    "phi" := "phi" + "w0c_11_24_5" * SIN(5 * 0.4 * "x") + "w0d_11_24_5" * COS(5 * 0.4 * "x");
    "phi" := "phi" + "w0c_11_24_6" * SIN(6 * 0.4 * "x") + "w0d_11_24_6" * COS(6 * 0.4 * "x");
    "acc" := "acc" + "phi";
    "x" := "feat_25";
    "phi" := "w0b_11_25" * "x" / (1.0 + EXP(-"x"));
    "phi" := "phi" + "w0c_11_25_1" * SIN(1 * 0.4 * "x") + "w0d_11_25_1" * COS(1 * 0.4 * "x");
    "phi" := "phi" + "w0c_11_25_2" * SIN(2 * 0.4 * "x") + "w0d_11_25_2" * COS(2 * 0.4 * "x");
    "phi" := "phi" + "w0c_11_25_3" * SIN(3 * 0.4 * "x") + "w0d_11_25_3" * COS(3 * 0.4 * "x");
    "phi" := "phi" + "w0c_11_25_4" * SIN(4 * 0.4 * "x") + "w0d_11_25_4" * COS(4 * 0.4 * "x");
    "phi" := "phi" + "w0c_11_25_5" * SIN(5 * 0.4 * "x") + "w0d_11_25_5" * COS(5 * 0.4 * "x");
    "phi" := "phi" + "w0c_11_25_6" * SIN(6 * 0.4 * "x") + "w0d_11_25_6" * COS(6 * 0.4 * "x");
    "acc" := "acc" + "phi";
    "x" := "feat_26";
    "phi" := "w0b_11_26" * "x" / (1.0 + EXP(-"x"));
    "phi" := "phi" + "w0c_11_26_1" * SIN(1 * 0.4 * "x") + "w0d_11_26_1" * COS(1 * 0.4 * "x");
    "phi" := "phi" + "w0c_11_26_2" * SIN(2 * 0.4 * "x") + "w0d_11_26_2" * COS(2 * 0.4 * "x");
    "phi" := "phi" + "w0c_11_26_3" * SIN(3 * 0.4 * "x") + "w0d_11_26_3" * COS(3 * 0.4 * "x");
    "phi" := "phi" + "w0c_11_26_4" * SIN(4 * 0.4 * "x") + "w0d_11_26_4" * COS(4 * 0.4 * "x");
    "phi" := "phi" + "w0c_11_26_5" * SIN(5 * 0.4 * "x") + "w0d_11_26_5" * COS(5 * 0.4 * "x");
    "phi" := "phi" + "w0c_11_26_6" * SIN(6 * 0.4 * "x") + "w0d_11_26_6" * COS(6 * 0.4 * "x");
    "acc" := "acc" + "phi";
    "x" := "feat_27";
    "phi" := "w0b_11_27" * "x" / (1.0 + EXP(-"x"));
    "phi" := "phi" + "w0c_11_27_1" * SIN(1 * 0.4 * "x") + "w0d_11_27_1" * COS(1 * 0.4 * "x");
    "phi" := "phi" + "w0c_11_27_2" * SIN(2 * 0.4 * "x") + "w0d_11_27_2" * COS(2 * 0.4 * "x");
    "phi" := "phi" + "w0c_11_27_3" * SIN(3 * 0.4 * "x") + "w0d_11_27_3" * COS(3 * 0.4 * "x");
    "phi" := "phi" + "w0c_11_27_4" * SIN(4 * 0.4 * "x") + "w0d_11_27_4" * COS(4 * 0.4 * "x");
    "phi" := "phi" + "w0c_11_27_5" * SIN(5 * 0.4 * "x") + "w0d_11_27_5" * COS(5 * 0.4 * "x");
    "phi" := "phi" + "w0c_11_27_6" * SIN(6 * 0.4 * "x") + "w0d_11_27_6" * COS(6 * 0.4 * "x");
    "acc" := "acc" + "phi";
    "x" := "feat_28";
    "phi" := "w0b_11_28" * "x" / (1.0 + EXP(-"x"));
    "phi" := "phi" + "w0c_11_28_1" * SIN(1 * 0.4 * "x") + "w0d_11_28_1" * COS(1 * 0.4 * "x");
    "phi" := "phi" + "w0c_11_28_2" * SIN(2 * 0.4 * "x") + "w0d_11_28_2" * COS(2 * 0.4 * "x");
    "phi" := "phi" + "w0c_11_28_3" * SIN(3 * 0.4 * "x") + "w0d_11_28_3" * COS(3 * 0.4 * "x");
    "phi" := "phi" + "w0c_11_28_4" * SIN(4 * 0.4 * "x") + "w0d_11_28_4" * COS(4 * 0.4 * "x");
    "phi" := "phi" + "w0c_11_28_5" * SIN(5 * 0.4 * "x") + "w0d_11_28_5" * COS(5 * 0.4 * "x");
    "phi" := "phi" + "w0c_11_28_6" * SIN(6 * 0.4 * "x") + "w0d_11_28_6" * COS(6 * 0.4 * "x");
    "acc" := "acc" + "phi";
    "h1_11" := "acc" + "b0_11";
    "acc" := 0.0;
    "x" := "feat_1";
    "phi" := "w0b_12_1" * "x" / (1.0 + EXP(-"x"));
    "phi" := "phi" + "w0c_12_1_1" * SIN(1 * 0.4 * "x") + "w0d_12_1_1" * COS(1 * 0.4 * "x");
    "phi" := "phi" + "w0c_12_1_2" * SIN(2 * 0.4 * "x") + "w0d_12_1_2" * COS(2 * 0.4 * "x");
    "phi" := "phi" + "w0c_12_1_3" * SIN(3 * 0.4 * "x") + "w0d_12_1_3" * COS(3 * 0.4 * "x");
    "phi" := "phi" + "w0c_12_1_4" * SIN(4 * 0.4 * "x") + "w0d_12_1_4" * COS(4 * 0.4 * "x");
    "phi" := "phi" + "w0c_12_1_5" * SIN(5 * 0.4 * "x") + "w0d_12_1_5" * COS(5 * 0.4 * "x");
    "phi" := "phi" + "w0c_12_1_6" * SIN(6 * 0.4 * "x") + "w0d_12_1_6" * COS(6 * 0.4 * "x");
    "acc" := "acc" + "phi";
    "x" := "feat_2";
    "phi" := "w0b_12_2" * "x" / (1.0 + EXP(-"x"));
    "phi" := "phi" + "w0c_12_2_1" * SIN(1 * 0.4 * "x") + "w0d_12_2_1" * COS(1 * 0.4 * "x");
    "phi" := "phi" + "w0c_12_2_2" * SIN(2 * 0.4 * "x") + "w0d_12_2_2" * COS(2 * 0.4 * "x");
    "phi" := "phi" + "w0c_12_2_3" * SIN(3 * 0.4 * "x") + "w0d_12_2_3" * COS(3 * 0.4 * "x");
    "phi" := "phi" + "w0c_12_2_4" * SIN(4 * 0.4 * "x") + "w0d_12_2_4" * COS(4 * 0.4 * "x");
    "phi" := "phi" + "w0c_12_2_5" * SIN(5 * 0.4 * "x") + "w0d_12_2_5" * COS(5 * 0.4 * "x");
    "phi" := "phi" + "w0c_12_2_6" * SIN(6 * 0.4 * "x") + "w0d_12_2_6" * COS(6 * 0.4 * "x");
    "acc" := "acc" + "phi";
    "x" := "feat_3";
    "phi" := "w0b_12_3" * "x" / (1.0 + EXP(-"x"));
    "phi" := "phi" + "w0c_12_3_1" * SIN(1 * 0.4 * "x") + "w0d_12_3_1" * COS(1 * 0.4 * "x");
    "phi" := "phi" + "w0c_12_3_2" * SIN(2 * 0.4 * "x") + "w0d_12_3_2" * COS(2 * 0.4 * "x");
    "phi" := "phi" + "w0c_12_3_3" * SIN(3 * 0.4 * "x") + "w0d_12_3_3" * COS(3 * 0.4 * "x");
    "phi" := "phi" + "w0c_12_3_4" * SIN(4 * 0.4 * "x") + "w0d_12_3_4" * COS(4 * 0.4 * "x");
    "phi" := "phi" + "w0c_12_3_5" * SIN(5 * 0.4 * "x") + "w0d_12_3_5" * COS(5 * 0.4 * "x");
    "phi" := "phi" + "w0c_12_3_6" * SIN(6 * 0.4 * "x") + "w0d_12_3_6" * COS(6 * 0.4 * "x");
    "acc" := "acc" + "phi";
    "x" := "feat_4";
    "phi" := "w0b_12_4" * "x" / (1.0 + EXP(-"x"));
    "phi" := "phi" + "w0c_12_4_1" * SIN(1 * 0.4 * "x") + "w0d_12_4_1" * COS(1 * 0.4 * "x");
    "phi" := "phi" + "w0c_12_4_2" * SIN(2 * 0.4 * "x") + "w0d_12_4_2" * COS(2 * 0.4 * "x");
    "phi" := "phi" + "w0c_12_4_3" * SIN(3 * 0.4 * "x") + "w0d_12_4_3" * COS(3 * 0.4 * "x");
    "phi" := "phi" + "w0c_12_4_4" * SIN(4 * 0.4 * "x") + "w0d_12_4_4" * COS(4 * 0.4 * "x");
    "phi" := "phi" + "w0c_12_4_5" * SIN(5 * 0.4 * "x") + "w0d_12_4_5" * COS(5 * 0.4 * "x");
    "phi" := "phi" + "w0c_12_4_6" * SIN(6 * 0.4 * "x") + "w0d_12_4_6" * COS(6 * 0.4 * "x");
    "acc" := "acc" + "phi";
    "x" := "feat_5";
    "phi" := "w0b_12_5" * "x" / (1.0 + EXP(-"x"));
    "phi" := "phi" + "w0c_12_5_1" * SIN(1 * 0.4 * "x") + "w0d_12_5_1" * COS(1 * 0.4 * "x");
    "phi" := "phi" + "w0c_12_5_2" * SIN(2 * 0.4 * "x") + "w0d_12_5_2" * COS(2 * 0.4 * "x");
    "phi" := "phi" + "w0c_12_5_3" * SIN(3 * 0.4 * "x") + "w0d_12_5_3" * COS(3 * 0.4 * "x");
    "phi" := "phi" + "w0c_12_5_4" * SIN(4 * 0.4 * "x") + "w0d_12_5_4" * COS(4 * 0.4 * "x");
    "phi" := "phi" + "w0c_12_5_5" * SIN(5 * 0.4 * "x") + "w0d_12_5_5" * COS(5 * 0.4 * "x");
    "phi" := "phi" + "w0c_12_5_6" * SIN(6 * 0.4 * "x") + "w0d_12_5_6" * COS(6 * 0.4 * "x");
    "acc" := "acc" + "phi";
    "x" := "feat_6";
    "phi" := "w0b_12_6" * "x" / (1.0 + EXP(-"x"));
    "phi" := "phi" + "w0c_12_6_1" * SIN(1 * 0.4 * "x") + "w0d_12_6_1" * COS(1 * 0.4 * "x");
    "phi" := "phi" + "w0c_12_6_2" * SIN(2 * 0.4 * "x") + "w0d_12_6_2" * COS(2 * 0.4 * "x");
    "phi" := "phi" + "w0c_12_6_3" * SIN(3 * 0.4 * "x") + "w0d_12_6_3" * COS(3 * 0.4 * "x");
    "phi" := "phi" + "w0c_12_6_4" * SIN(4 * 0.4 * "x") + "w0d_12_6_4" * COS(4 * 0.4 * "x");
    "phi" := "phi" + "w0c_12_6_5" * SIN(5 * 0.4 * "x") + "w0d_12_6_5" * COS(5 * 0.4 * "x");
    "phi" := "phi" + "w0c_12_6_6" * SIN(6 * 0.4 * "x") + "w0d_12_6_6" * COS(6 * 0.4 * "x");
    "acc" := "acc" + "phi";
    "x" := "feat_7";
    "phi" := "w0b_12_7" * "x" / (1.0 + EXP(-"x"));
    "phi" := "phi" + "w0c_12_7_1" * SIN(1 * 0.4 * "x") + "w0d_12_7_1" * COS(1 * 0.4 * "x");
    "phi" := "phi" + "w0c_12_7_2" * SIN(2 * 0.4 * "x") + "w0d_12_7_2" * COS(2 * 0.4 * "x");
    "phi" := "phi" + "w0c_12_7_3" * SIN(3 * 0.4 * "x") + "w0d_12_7_3" * COS(3 * 0.4 * "x");
    "phi" := "phi" + "w0c_12_7_4" * SIN(4 * 0.4 * "x") + "w0d_12_7_4" * COS(4 * 0.4 * "x");
    "phi" := "phi" + "w0c_12_7_5" * SIN(5 * 0.4 * "x") + "w0d_12_7_5" * COS(5 * 0.4 * "x");
    "phi" := "phi" + "w0c_12_7_6" * SIN(6 * 0.4 * "x") + "w0d_12_7_6" * COS(6 * 0.4 * "x");
    "acc" := "acc" + "phi";
    "x" := "feat_8";
    "phi" := "w0b_12_8" * "x" / (1.0 + EXP(-"x"));
    "phi" := "phi" + "w0c_12_8_1" * SIN(1 * 0.4 * "x") + "w0d_12_8_1" * COS(1 * 0.4 * "x");
    "phi" := "phi" + "w0c_12_8_2" * SIN(2 * 0.4 * "x") + "w0d_12_8_2" * COS(2 * 0.4 * "x");
    "phi" := "phi" + "w0c_12_8_3" * SIN(3 * 0.4 * "x") + "w0d_12_8_3" * COS(3 * 0.4 * "x");
    "phi" := "phi" + "w0c_12_8_4" * SIN(4 * 0.4 * "x") + "w0d_12_8_4" * COS(4 * 0.4 * "x");
    "phi" := "phi" + "w0c_12_8_5" * SIN(5 * 0.4 * "x") + "w0d_12_8_5" * COS(5 * 0.4 * "x");
    "phi" := "phi" + "w0c_12_8_6" * SIN(6 * 0.4 * "x") + "w0d_12_8_6" * COS(6 * 0.4 * "x");
    "acc" := "acc" + "phi";
    "x" := "feat_9";
    "phi" := "w0b_12_9" * "x" / (1.0 + EXP(-"x"));
    "phi" := "phi" + "w0c_12_9_1" * SIN(1 * 0.4 * "x") + "w0d_12_9_1" * COS(1 * 0.4 * "x");
    "phi" := "phi" + "w0c_12_9_2" * SIN(2 * 0.4 * "x") + "w0d_12_9_2" * COS(2 * 0.4 * "x");
    "phi" := "phi" + "w0c_12_9_3" * SIN(3 * 0.4 * "x") + "w0d_12_9_3" * COS(3 * 0.4 * "x");
    "phi" := "phi" + "w0c_12_9_4" * SIN(4 * 0.4 * "x") + "w0d_12_9_4" * COS(4 * 0.4 * "x");
    "phi" := "phi" + "w0c_12_9_5" * SIN(5 * 0.4 * "x") + "w0d_12_9_5" * COS(5 * 0.4 * "x");
    "phi" := "phi" + "w0c_12_9_6" * SIN(6 * 0.4 * "x") + "w0d_12_9_6" * COS(6 * 0.4 * "x");
    "acc" := "acc" + "phi";
    "x" := "feat_10";
    "phi" := "w0b_12_10" * "x" / (1.0 + EXP(-"x"));
    "phi" := "phi" + "w0c_12_10_1" * SIN(1 * 0.4 * "x") + "w0d_12_10_1" * COS(1 * 0.4 * "x");
    "phi" := "phi" + "w0c_12_10_2" * SIN(2 * 0.4 * "x") + "w0d_12_10_2" * COS(2 * 0.4 * "x");
    "phi" := "phi" + "w0c_12_10_3" * SIN(3 * 0.4 * "x") + "w0d_12_10_3" * COS(3 * 0.4 * "x");
    "phi" := "phi" + "w0c_12_10_4" * SIN(4 * 0.4 * "x") + "w0d_12_10_4" * COS(4 * 0.4 * "x");
    "phi" := "phi" + "w0c_12_10_5" * SIN(5 * 0.4 * "x") + "w0d_12_10_5" * COS(5 * 0.4 * "x");
    "phi" := "phi" + "w0c_12_10_6" * SIN(6 * 0.4 * "x") + "w0d_12_10_6" * COS(6 * 0.4 * "x");
    "acc" := "acc" + "phi";
    "x" := "feat_11";
    "phi" := "w0b_12_11" * "x" / (1.0 + EXP(-"x"));
    "phi" := "phi" + "w0c_12_11_1" * SIN(1 * 0.4 * "x") + "w0d_12_11_1" * COS(1 * 0.4 * "x");
    "phi" := "phi" + "w0c_12_11_2" * SIN(2 * 0.4 * "x") + "w0d_12_11_2" * COS(2 * 0.4 * "x");
    "phi" := "phi" + "w0c_12_11_3" * SIN(3 * 0.4 * "x") + "w0d_12_11_3" * COS(3 * 0.4 * "x");
    "phi" := "phi" + "w0c_12_11_4" * SIN(4 * 0.4 * "x") + "w0d_12_11_4" * COS(4 * 0.4 * "x");
    "phi" := "phi" + "w0c_12_11_5" * SIN(5 * 0.4 * "x") + "w0d_12_11_5" * COS(5 * 0.4 * "x");
    "phi" := "phi" + "w0c_12_11_6" * SIN(6 * 0.4 * "x") + "w0d_12_11_6" * COS(6 * 0.4 * "x");
    "acc" := "acc" + "phi";
    "x" := "feat_12";
    "phi" := "w0b_12_12" * "x" / (1.0 + EXP(-"x"));
    "phi" := "phi" + "w0c_12_12_1" * SIN(1 * 0.4 * "x") + "w0d_12_12_1" * COS(1 * 0.4 * "x");
    "phi" := "phi" + "w0c_12_12_2" * SIN(2 * 0.4 * "x") + "w0d_12_12_2" * COS(2 * 0.4 * "x");
    "phi" := "phi" + "w0c_12_12_3" * SIN(3 * 0.4 * "x") + "w0d_12_12_3" * COS(3 * 0.4 * "x");
    "phi" := "phi" + "w0c_12_12_4" * SIN(4 * 0.4 * "x") + "w0d_12_12_4" * COS(4 * 0.4 * "x");
    "phi" := "phi" + "w0c_12_12_5" * SIN(5 * 0.4 * "x") + "w0d_12_12_5" * COS(5 * 0.4 * "x");
    "phi" := "phi" + "w0c_12_12_6" * SIN(6 * 0.4 * "x") + "w0d_12_12_6" * COS(6 * 0.4 * "x");
    "acc" := "acc" + "phi";
    "x" := "feat_13";
    "phi" := "w0b_12_13" * "x" / (1.0 + EXP(-"x"));
    "phi" := "phi" + "w0c_12_13_1" * SIN(1 * 0.4 * "x") + "w0d_12_13_1" * COS(1 * 0.4 * "x");
    "phi" := "phi" + "w0c_12_13_2" * SIN(2 * 0.4 * "x") + "w0d_12_13_2" * COS(2 * 0.4 * "x");
    "phi" := "phi" + "w0c_12_13_3" * SIN(3 * 0.4 * "x") + "w0d_12_13_3" * COS(3 * 0.4 * "x");
    "phi" := "phi" + "w0c_12_13_4" * SIN(4 * 0.4 * "x") + "w0d_12_13_4" * COS(4 * 0.4 * "x");
    "phi" := "phi" + "w0c_12_13_5" * SIN(5 * 0.4 * "x") + "w0d_12_13_5" * COS(5 * 0.4 * "x");
    "phi" := "phi" + "w0c_12_13_6" * SIN(6 * 0.4 * "x") + "w0d_12_13_6" * COS(6 * 0.4 * "x");
    "acc" := "acc" + "phi";
    "x" := "feat_14";
    "phi" := "w0b_12_14" * "x" / (1.0 + EXP(-"x"));
    "phi" := "phi" + "w0c_12_14_1" * SIN(1 * 0.4 * "x") + "w0d_12_14_1" * COS(1 * 0.4 * "x");
    "phi" := "phi" + "w0c_12_14_2" * SIN(2 * 0.4 * "x") + "w0d_12_14_2" * COS(2 * 0.4 * "x");
    "phi" := "phi" + "w0c_12_14_3" * SIN(3 * 0.4 * "x") + "w0d_12_14_3" * COS(3 * 0.4 * "x");
    "phi" := "phi" + "w0c_12_14_4" * SIN(4 * 0.4 * "x") + "w0d_12_14_4" * COS(4 * 0.4 * "x");
    "phi" := "phi" + "w0c_12_14_5" * SIN(5 * 0.4 * "x") + "w0d_12_14_5" * COS(5 * 0.4 * "x");
    "phi" := "phi" + "w0c_12_14_6" * SIN(6 * 0.4 * "x") + "w0d_12_14_6" * COS(6 * 0.4 * "x");
    "acc" := "acc" + "phi";
    "x" := "feat_15";
    "phi" := "w0b_12_15" * "x" / (1.0 + EXP(-"x"));
    "phi" := "phi" + "w0c_12_15_1" * SIN(1 * 0.4 * "x") + "w0d_12_15_1" * COS(1 * 0.4 * "x");
    "phi" := "phi" + "w0c_12_15_2" * SIN(2 * 0.4 * "x") + "w0d_12_15_2" * COS(2 * 0.4 * "x");
    "phi" := "phi" + "w0c_12_15_3" * SIN(3 * 0.4 * "x") + "w0d_12_15_3" * COS(3 * 0.4 * "x");
    "phi" := "phi" + "w0c_12_15_4" * SIN(4 * 0.4 * "x") + "w0d_12_15_4" * COS(4 * 0.4 * "x");
    "phi" := "phi" + "w0c_12_15_5" * SIN(5 * 0.4 * "x") + "w0d_12_15_5" * COS(5 * 0.4 * "x");
    "phi" := "phi" + "w0c_12_15_6" * SIN(6 * 0.4 * "x") + "w0d_12_15_6" * COS(6 * 0.4 * "x");
    "acc" := "acc" + "phi";
    "x" := "feat_16";
    "phi" := "w0b_12_16" * "x" / (1.0 + EXP(-"x"));
    "phi" := "phi" + "w0c_12_16_1" * SIN(1 * 0.4 * "x") + "w0d_12_16_1" * COS(1 * 0.4 * "x");
    "phi" := "phi" + "w0c_12_16_2" * SIN(2 * 0.4 * "x") + "w0d_12_16_2" * COS(2 * 0.4 * "x");
    "phi" := "phi" + "w0c_12_16_3" * SIN(3 * 0.4 * "x") + "w0d_12_16_3" * COS(3 * 0.4 * "x");
    "phi" := "phi" + "w0c_12_16_4" * SIN(4 * 0.4 * "x") + "w0d_12_16_4" * COS(4 * 0.4 * "x");
    "phi" := "phi" + "w0c_12_16_5" * SIN(5 * 0.4 * "x") + "w0d_12_16_5" * COS(5 * 0.4 * "x");
    "phi" := "phi" + "w0c_12_16_6" * SIN(6 * 0.4 * "x") + "w0d_12_16_6" * COS(6 * 0.4 * "x");
    "acc" := "acc" + "phi";
    "x" := "feat_17";
    "phi" := "w0b_12_17" * "x" / (1.0 + EXP(-"x"));
    "phi" := "phi" + "w0c_12_17_1" * SIN(1 * 0.4 * "x") + "w0d_12_17_1" * COS(1 * 0.4 * "x");
    "phi" := "phi" + "w0c_12_17_2" * SIN(2 * 0.4 * "x") + "w0d_12_17_2" * COS(2 * 0.4 * "x");
    "phi" := "phi" + "w0c_12_17_3" * SIN(3 * 0.4 * "x") + "w0d_12_17_3" * COS(3 * 0.4 * "x");
    "phi" := "phi" + "w0c_12_17_4" * SIN(4 * 0.4 * "x") + "w0d_12_17_4" * COS(4 * 0.4 * "x");
    "phi" := "phi" + "w0c_12_17_5" * SIN(5 * 0.4 * "x") + "w0d_12_17_5" * COS(5 * 0.4 * "x");
    "phi" := "phi" + "w0c_12_17_6" * SIN(6 * 0.4 * "x") + "w0d_12_17_6" * COS(6 * 0.4 * "x");
    "acc" := "acc" + "phi";
    "x" := "feat_18";
    "phi" := "w0b_12_18" * "x" / (1.0 + EXP(-"x"));
    "phi" := "phi" + "w0c_12_18_1" * SIN(1 * 0.4 * "x") + "w0d_12_18_1" * COS(1 * 0.4 * "x");
    "phi" := "phi" + "w0c_12_18_2" * SIN(2 * 0.4 * "x") + "w0d_12_18_2" * COS(2 * 0.4 * "x");
    "phi" := "phi" + "w0c_12_18_3" * SIN(3 * 0.4 * "x") + "w0d_12_18_3" * COS(3 * 0.4 * "x");
    "phi" := "phi" + "w0c_12_18_4" * SIN(4 * 0.4 * "x") + "w0d_12_18_4" * COS(4 * 0.4 * "x");
    "phi" := "phi" + "w0c_12_18_5" * SIN(5 * 0.4 * "x") + "w0d_12_18_5" * COS(5 * 0.4 * "x");
    "phi" := "phi" + "w0c_12_18_6" * SIN(6 * 0.4 * "x") + "w0d_12_18_6" * COS(6 * 0.4 * "x");
    "acc" := "acc" + "phi";
    "x" := "feat_19";
    "phi" := "w0b_12_19" * "x" / (1.0 + EXP(-"x"));
    "phi" := "phi" + "w0c_12_19_1" * SIN(1 * 0.4 * "x") + "w0d_12_19_1" * COS(1 * 0.4 * "x");
    "phi" := "phi" + "w0c_12_19_2" * SIN(2 * 0.4 * "x") + "w0d_12_19_2" * COS(2 * 0.4 * "x");
    "phi" := "phi" + "w0c_12_19_3" * SIN(3 * 0.4 * "x") + "w0d_12_19_3" * COS(3 * 0.4 * "x");
    "phi" := "phi" + "w0c_12_19_4" * SIN(4 * 0.4 * "x") + "w0d_12_19_4" * COS(4 * 0.4 * "x");
    "phi" := "phi" + "w0c_12_19_5" * SIN(5 * 0.4 * "x") + "w0d_12_19_5" * COS(5 * 0.4 * "x");
    "phi" := "phi" + "w0c_12_19_6" * SIN(6 * 0.4 * "x") + "w0d_12_19_6" * COS(6 * 0.4 * "x");
    "acc" := "acc" + "phi";
    "x" := "feat_20";
    "phi" := "w0b_12_20" * "x" / (1.0 + EXP(-"x"));
    "phi" := "phi" + "w0c_12_20_1" * SIN(1 * 0.4 * "x") + "w0d_12_20_1" * COS(1 * 0.4 * "x");
    "phi" := "phi" + "w0c_12_20_2" * SIN(2 * 0.4 * "x") + "w0d_12_20_2" * COS(2 * 0.4 * "x");
    "phi" := "phi" + "w0c_12_20_3" * SIN(3 * 0.4 * "x") + "w0d_12_20_3" * COS(3 * 0.4 * "x");
    "phi" := "phi" + "w0c_12_20_4" * SIN(4 * 0.4 * "x") + "w0d_12_20_4" * COS(4 * 0.4 * "x");
    "phi" := "phi" + "w0c_12_20_5" * SIN(5 * 0.4 * "x") + "w0d_12_20_5" * COS(5 * 0.4 * "x");
    "phi" := "phi" + "w0c_12_20_6" * SIN(6 * 0.4 * "x") + "w0d_12_20_6" * COS(6 * 0.4 * "x");
    "acc" := "acc" + "phi";
    "x" := "feat_21";
    "phi" := "w0b_12_21" * "x" / (1.0 + EXP(-"x"));
    "phi" := "phi" + "w0c_12_21_1" * SIN(1 * 0.4 * "x") + "w0d_12_21_1" * COS(1 * 0.4 * "x");
    "phi" := "phi" + "w0c_12_21_2" * SIN(2 * 0.4 * "x") + "w0d_12_21_2" * COS(2 * 0.4 * "x");
    "phi" := "phi" + "w0c_12_21_3" * SIN(3 * 0.4 * "x") + "w0d_12_21_3" * COS(3 * 0.4 * "x");
    "phi" := "phi" + "w0c_12_21_4" * SIN(4 * 0.4 * "x") + "w0d_12_21_4" * COS(4 * 0.4 * "x");
    "phi" := "phi" + "w0c_12_21_5" * SIN(5 * 0.4 * "x") + "w0d_12_21_5" * COS(5 * 0.4 * "x");
    "phi" := "phi" + "w0c_12_21_6" * SIN(6 * 0.4 * "x") + "w0d_12_21_6" * COS(6 * 0.4 * "x");
    "acc" := "acc" + "phi";
    "x" := "feat_22";
    "phi" := "w0b_12_22" * "x" / (1.0 + EXP(-"x"));
    "phi" := "phi" + "w0c_12_22_1" * SIN(1 * 0.4 * "x") + "w0d_12_22_1" * COS(1 * 0.4 * "x");
    "phi" := "phi" + "w0c_12_22_2" * SIN(2 * 0.4 * "x") + "w0d_12_22_2" * COS(2 * 0.4 * "x");
    "phi" := "phi" + "w0c_12_22_3" * SIN(3 * 0.4 * "x") + "w0d_12_22_3" * COS(3 * 0.4 * "x");
    "phi" := "phi" + "w0c_12_22_4" * SIN(4 * 0.4 * "x") + "w0d_12_22_4" * COS(4 * 0.4 * "x");
    "phi" := "phi" + "w0c_12_22_5" * SIN(5 * 0.4 * "x") + "w0d_12_22_5" * COS(5 * 0.4 * "x");
    "phi" := "phi" + "w0c_12_22_6" * SIN(6 * 0.4 * "x") + "w0d_12_22_6" * COS(6 * 0.4 * "x");
    "acc" := "acc" + "phi";
    "x" := "feat_23";
    "phi" := "w0b_12_23" * "x" / (1.0 + EXP(-"x"));
    "phi" := "phi" + "w0c_12_23_1" * SIN(1 * 0.4 * "x") + "w0d_12_23_1" * COS(1 * 0.4 * "x");
    "phi" := "phi" + "w0c_12_23_2" * SIN(2 * 0.4 * "x") + "w0d_12_23_2" * COS(2 * 0.4 * "x");
    "phi" := "phi" + "w0c_12_23_3" * SIN(3 * 0.4 * "x") + "w0d_12_23_3" * COS(3 * 0.4 * "x");
    "phi" := "phi" + "w0c_12_23_4" * SIN(4 * 0.4 * "x") + "w0d_12_23_4" * COS(4 * 0.4 * "x");
    "phi" := "phi" + "w0c_12_23_5" * SIN(5 * 0.4 * "x") + "w0d_12_23_5" * COS(5 * 0.4 * "x");
    "phi" := "phi" + "w0c_12_23_6" * SIN(6 * 0.4 * "x") + "w0d_12_23_6" * COS(6 * 0.4 * "x");
    "acc" := "acc" + "phi";
    "x" := "feat_24";
    "phi" := "w0b_12_24" * "x" / (1.0 + EXP(-"x"));
    "phi" := "phi" + "w0c_12_24_1" * SIN(1 * 0.4 * "x") + "w0d_12_24_1" * COS(1 * 0.4 * "x");
    "phi" := "phi" + "w0c_12_24_2" * SIN(2 * 0.4 * "x") + "w0d_12_24_2" * COS(2 * 0.4 * "x");
    "phi" := "phi" + "w0c_12_24_3" * SIN(3 * 0.4 * "x") + "w0d_12_24_3" * COS(3 * 0.4 * "x");
    "phi" := "phi" + "w0c_12_24_4" * SIN(4 * 0.4 * "x") + "w0d_12_24_4" * COS(4 * 0.4 * "x");
    "phi" := "phi" + "w0c_12_24_5" * SIN(5 * 0.4 * "x") + "w0d_12_24_5" * COS(5 * 0.4 * "x");
    "phi" := "phi" + "w0c_12_24_6" * SIN(6 * 0.4 * "x") + "w0d_12_24_6" * COS(6 * 0.4 * "x");
    "acc" := "acc" + "phi";
    "x" := "feat_25";
    "phi" := "w0b_12_25" * "x" / (1.0 + EXP(-"x"));
    "phi" := "phi" + "w0c_12_25_1" * SIN(1 * 0.4 * "x") + "w0d_12_25_1" * COS(1 * 0.4 * "x");
    "phi" := "phi" + "w0c_12_25_2" * SIN(2 * 0.4 * "x") + "w0d_12_25_2" * COS(2 * 0.4 * "x");
    "phi" := "phi" + "w0c_12_25_3" * SIN(3 * 0.4 * "x") + "w0d_12_25_3" * COS(3 * 0.4 * "x");
    "phi" := "phi" + "w0c_12_25_4" * SIN(4 * 0.4 * "x") + "w0d_12_25_4" * COS(4 * 0.4 * "x");
    "phi" := "phi" + "w0c_12_25_5" * SIN(5 * 0.4 * "x") + "w0d_12_25_5" * COS(5 * 0.4 * "x");
    "phi" := "phi" + "w0c_12_25_6" * SIN(6 * 0.4 * "x") + "w0d_12_25_6" * COS(6 * 0.4 * "x");
    "acc" := "acc" + "phi";
    "x" := "feat_26";
    "phi" := "w0b_12_26" * "x" / (1.0 + EXP(-"x"));
    "phi" := "phi" + "w0c_12_26_1" * SIN(1 * 0.4 * "x") + "w0d_12_26_1" * COS(1 * 0.4 * "x");
    "phi" := "phi" + "w0c_12_26_2" * SIN(2 * 0.4 * "x") + "w0d_12_26_2" * COS(2 * 0.4 * "x");
    "phi" := "phi" + "w0c_12_26_3" * SIN(3 * 0.4 * "x") + "w0d_12_26_3" * COS(3 * 0.4 * "x");
    "phi" := "phi" + "w0c_12_26_4" * SIN(4 * 0.4 * "x") + "w0d_12_26_4" * COS(4 * 0.4 * "x");
    "phi" := "phi" + "w0c_12_26_5" * SIN(5 * 0.4 * "x") + "w0d_12_26_5" * COS(5 * 0.4 * "x");
    "phi" := "phi" + "w0c_12_26_6" * SIN(6 * 0.4 * "x") + "w0d_12_26_6" * COS(6 * 0.4 * "x");
    "acc" := "acc" + "phi";
    "x" := "feat_27";
    "phi" := "w0b_12_27" * "x" / (1.0 + EXP(-"x"));
    "phi" := "phi" + "w0c_12_27_1" * SIN(1 * 0.4 * "x") + "w0d_12_27_1" * COS(1 * 0.4 * "x");
    "phi" := "phi" + "w0c_12_27_2" * SIN(2 * 0.4 * "x") + "w0d_12_27_2" * COS(2 * 0.4 * "x");
    "phi" := "phi" + "w0c_12_27_3" * SIN(3 * 0.4 * "x") + "w0d_12_27_3" * COS(3 * 0.4 * "x");
    "phi" := "phi" + "w0c_12_27_4" * SIN(4 * 0.4 * "x") + "w0d_12_27_4" * COS(4 * 0.4 * "x");
    "phi" := "phi" + "w0c_12_27_5" * SIN(5 * 0.4 * "x") + "w0d_12_27_5" * COS(5 * 0.4 * "x");
    "phi" := "phi" + "w0c_12_27_6" * SIN(6 * 0.4 * "x") + "w0d_12_27_6" * COS(6 * 0.4 * "x");
    "acc" := "acc" + "phi";
    "x" := "feat_28";
    "phi" := "w0b_12_28" * "x" / (1.0 + EXP(-"x"));
    "phi" := "phi" + "w0c_12_28_1" * SIN(1 * 0.4 * "x") + "w0d_12_28_1" * COS(1 * 0.4 * "x");
    "phi" := "phi" + "w0c_12_28_2" * SIN(2 * 0.4 * "x") + "w0d_12_28_2" * COS(2 * 0.4 * "x");
    "phi" := "phi" + "w0c_12_28_3" * SIN(3 * 0.4 * "x") + "w0d_12_28_3" * COS(3 * 0.4 * "x");
    "phi" := "phi" + "w0c_12_28_4" * SIN(4 * 0.4 * "x") + "w0d_12_28_4" * COS(4 * 0.4 * "x");
    "phi" := "phi" + "w0c_12_28_5" * SIN(5 * 0.4 * "x") + "w0d_12_28_5" * COS(5 * 0.4 * "x");
    "phi" := "phi" + "w0c_12_28_6" * SIN(6 * 0.4 * "x") + "w0d_12_28_6" * COS(6 * 0.4 * "x");
    "acc" := "acc" + "phi";
    "h1_12" := "acc" + "b0_12";
    "acc" := 0.0;
    "x" := "feat_1";
    "phi" := "w0b_13_1" * "x" / (1.0 + EXP(-"x"));
    "phi" := "phi" + "w0c_13_1_1" * SIN(1 * 0.4 * "x") + "w0d_13_1_1" * COS(1 * 0.4 * "x");
    "phi" := "phi" + "w0c_13_1_2" * SIN(2 * 0.4 * "x") + "w0d_13_1_2" * COS(2 * 0.4 * "x");
    "phi" := "phi" + "w0c_13_1_3" * SIN(3 * 0.4 * "x") + "w0d_13_1_3" * COS(3 * 0.4 * "x");
    "phi" := "phi" + "w0c_13_1_4" * SIN(4 * 0.4 * "x") + "w0d_13_1_4" * COS(4 * 0.4 * "x");
    "phi" := "phi" + "w0c_13_1_5" * SIN(5 * 0.4 * "x") + "w0d_13_1_5" * COS(5 * 0.4 * "x");
    "phi" := "phi" + "w0c_13_1_6" * SIN(6 * 0.4 * "x") + "w0d_13_1_6" * COS(6 * 0.4 * "x");
    "acc" := "acc" + "phi";
    "x" := "feat_2";
    "phi" := "w0b_13_2" * "x" / (1.0 + EXP(-"x"));
    "phi" := "phi" + "w0c_13_2_1" * SIN(1 * 0.4 * "x") + "w0d_13_2_1" * COS(1 * 0.4 * "x");
    "phi" := "phi" + "w0c_13_2_2" * SIN(2 * 0.4 * "x") + "w0d_13_2_2" * COS(2 * 0.4 * "x");
    "phi" := "phi" + "w0c_13_2_3" * SIN(3 * 0.4 * "x") + "w0d_13_2_3" * COS(3 * 0.4 * "x");
    "phi" := "phi" + "w0c_13_2_4" * SIN(4 * 0.4 * "x") + "w0d_13_2_4" * COS(4 * 0.4 * "x");
    "phi" := "phi" + "w0c_13_2_5" * SIN(5 * 0.4 * "x") + "w0d_13_2_5" * COS(5 * 0.4 * "x");
    "phi" := "phi" + "w0c_13_2_6" * SIN(6 * 0.4 * "x") + "w0d_13_2_6" * COS(6 * 0.4 * "x");
    "acc" := "acc" + "phi";
    "x" := "feat_3";
    "phi" := "w0b_13_3" * "x" / (1.0 + EXP(-"x"));
    "phi" := "phi" + "w0c_13_3_1" * SIN(1 * 0.4 * "x") + "w0d_13_3_1" * COS(1 * 0.4 * "x");
    "phi" := "phi" + "w0c_13_3_2" * SIN(2 * 0.4 * "x") + "w0d_13_3_2" * COS(2 * 0.4 * "x");
    "phi" := "phi" + "w0c_13_3_3" * SIN(3 * 0.4 * "x") + "w0d_13_3_3" * COS(3 * 0.4 * "x");
    "phi" := "phi" + "w0c_13_3_4" * SIN(4 * 0.4 * "x") + "w0d_13_3_4" * COS(4 * 0.4 * "x");
    "phi" := "phi" + "w0c_13_3_5" * SIN(5 * 0.4 * "x") + "w0d_13_3_5" * COS(5 * 0.4 * "x");
    "phi" := "phi" + "w0c_13_3_6" * SIN(6 * 0.4 * "x") + "w0d_13_3_6" * COS(6 * 0.4 * "x");
    "acc" := "acc" + "phi";
    "x" := "feat_4";
    "phi" := "w0b_13_4" * "x" / (1.0 + EXP(-"x"));
    "phi" := "phi" + "w0c_13_4_1" * SIN(1 * 0.4 * "x") + "w0d_13_4_1" * COS(1 * 0.4 * "x");
    "phi" := "phi" + "w0c_13_4_2" * SIN(2 * 0.4 * "x") + "w0d_13_4_2" * COS(2 * 0.4 * "x");
    "phi" := "phi" + "w0c_13_4_3" * SIN(3 * 0.4 * "x") + "w0d_13_4_3" * COS(3 * 0.4 * "x");
    "phi" := "phi" + "w0c_13_4_4" * SIN(4 * 0.4 * "x") + "w0d_13_4_4" * COS(4 * 0.4 * "x");
    "phi" := "phi" + "w0c_13_4_5" * SIN(5 * 0.4 * "x") + "w0d_13_4_5" * COS(5 * 0.4 * "x");
    "phi" := "phi" + "w0c_13_4_6" * SIN(6 * 0.4 * "x") + "w0d_13_4_6" * COS(6 * 0.4 * "x");
    "acc" := "acc" + "phi";
    "x" := "feat_5";
    "phi" := "w0b_13_5" * "x" / (1.0 + EXP(-"x"));
    "phi" := "phi" + "w0c_13_5_1" * SIN(1 * 0.4 * "x") + "w0d_13_5_1" * COS(1 * 0.4 * "x");
    "phi" := "phi" + "w0c_13_5_2" * SIN(2 * 0.4 * "x") + "w0d_13_5_2" * COS(2 * 0.4 * "x");
    "phi" := "phi" + "w0c_13_5_3" * SIN(3 * 0.4 * "x") + "w0d_13_5_3" * COS(3 * 0.4 * "x");
    "phi" := "phi" + "w0c_13_5_4" * SIN(4 * 0.4 * "x") + "w0d_13_5_4" * COS(4 * 0.4 * "x");
    "phi" := "phi" + "w0c_13_5_5" * SIN(5 * 0.4 * "x") + "w0d_13_5_5" * COS(5 * 0.4 * "x");
    "phi" := "phi" + "w0c_13_5_6" * SIN(6 * 0.4 * "x") + "w0d_13_5_6" * COS(6 * 0.4 * "x");
    "acc" := "acc" + "phi";
    "x" := "feat_6";
    "phi" := "w0b_13_6" * "x" / (1.0 + EXP(-"x"));
    "phi" := "phi" + "w0c_13_6_1" * SIN(1 * 0.4 * "x") + "w0d_13_6_1" * COS(1 * 0.4 * "x");
    "phi" := "phi" + "w0c_13_6_2" * SIN(2 * 0.4 * "x") + "w0d_13_6_2" * COS(2 * 0.4 * "x");
    "phi" := "phi" + "w0c_13_6_3" * SIN(3 * 0.4 * "x") + "w0d_13_6_3" * COS(3 * 0.4 * "x");
    "phi" := "phi" + "w0c_13_6_4" * SIN(4 * 0.4 * "x") + "w0d_13_6_4" * COS(4 * 0.4 * "x");
    "phi" := "phi" + "w0c_13_6_5" * SIN(5 * 0.4 * "x") + "w0d_13_6_5" * COS(5 * 0.4 * "x");
    "phi" := "phi" + "w0c_13_6_6" * SIN(6 * 0.4 * "x") + "w0d_13_6_6" * COS(6 * 0.4 * "x");
    "acc" := "acc" + "phi";
    "x" := "feat_7";
    "phi" := "w0b_13_7" * "x" / (1.0 + EXP(-"x"));
    "phi" := "phi" + "w0c_13_7_1" * SIN(1 * 0.4 * "x") + "w0d_13_7_1" * COS(1 * 0.4 * "x");
    "phi" := "phi" + "w0c_13_7_2" * SIN(2 * 0.4 * "x") + "w0d_13_7_2" * COS(2 * 0.4 * "x");
    "phi" := "phi" + "w0c_13_7_3" * SIN(3 * 0.4 * "x") + "w0d_13_7_3" * COS(3 * 0.4 * "x");
    "phi" := "phi" + "w0c_13_7_4" * SIN(4 * 0.4 * "x") + "w0d_13_7_4" * COS(4 * 0.4 * "x");
    "phi" := "phi" + "w0c_13_7_5" * SIN(5 * 0.4 * "x") + "w0d_13_7_5" * COS(5 * 0.4 * "x");
    "phi" := "phi" + "w0c_13_7_6" * SIN(6 * 0.4 * "x") + "w0d_13_7_6" * COS(6 * 0.4 * "x");
    "acc" := "acc" + "phi";
    "x" := "feat_8";
    "phi" := "w0b_13_8" * "x" / (1.0 + EXP(-"x"));
    "phi" := "phi" + "w0c_13_8_1" * SIN(1 * 0.4 * "x") + "w0d_13_8_1" * COS(1 * 0.4 * "x");
    "phi" := "phi" + "w0c_13_8_2" * SIN(2 * 0.4 * "x") + "w0d_13_8_2" * COS(2 * 0.4 * "x");
    "phi" := "phi" + "w0c_13_8_3" * SIN(3 * 0.4 * "x") + "w0d_13_8_3" * COS(3 * 0.4 * "x");
    "phi" := "phi" + "w0c_13_8_4" * SIN(4 * 0.4 * "x") + "w0d_13_8_4" * COS(4 * 0.4 * "x");
    "phi" := "phi" + "w0c_13_8_5" * SIN(5 * 0.4 * "x") + "w0d_13_8_5" * COS(5 * 0.4 * "x");
    "phi" := "phi" + "w0c_13_8_6" * SIN(6 * 0.4 * "x") + "w0d_13_8_6" * COS(6 * 0.4 * "x");
    "acc" := "acc" + "phi";
    "x" := "feat_9";
    "phi" := "w0b_13_9" * "x" / (1.0 + EXP(-"x"));
    "phi" := "phi" + "w0c_13_9_1" * SIN(1 * 0.4 * "x") + "w0d_13_9_1" * COS(1 * 0.4 * "x");
    "phi" := "phi" + "w0c_13_9_2" * SIN(2 * 0.4 * "x") + "w0d_13_9_2" * COS(2 * 0.4 * "x");
    "phi" := "phi" + "w0c_13_9_3" * SIN(3 * 0.4 * "x") + "w0d_13_9_3" * COS(3 * 0.4 * "x");
    "phi" := "phi" + "w0c_13_9_4" * SIN(4 * 0.4 * "x") + "w0d_13_9_4" * COS(4 * 0.4 * "x");
    "phi" := "phi" + "w0c_13_9_5" * SIN(5 * 0.4 * "x") + "w0d_13_9_5" * COS(5 * 0.4 * "x");
    "phi" := "phi" + "w0c_13_9_6" * SIN(6 * 0.4 * "x") + "w0d_13_9_6" * COS(6 * 0.4 * "x");
    "acc" := "acc" + "phi";
    "x" := "feat_10";
    "phi" := "w0b_13_10" * "x" / (1.0 + EXP(-"x"));
    "phi" := "phi" + "w0c_13_10_1" * SIN(1 * 0.4 * "x") + "w0d_13_10_1" * COS(1 * 0.4 * "x");
    "phi" := "phi" + "w0c_13_10_2" * SIN(2 * 0.4 * "x") + "w0d_13_10_2" * COS(2 * 0.4 * "x");
    "phi" := "phi" + "w0c_13_10_3" * SIN(3 * 0.4 * "x") + "w0d_13_10_3" * COS(3 * 0.4 * "x");
    "phi" := "phi" + "w0c_13_10_4" * SIN(4 * 0.4 * "x") + "w0d_13_10_4" * COS(4 * 0.4 * "x");
    "phi" := "phi" + "w0c_13_10_5" * SIN(5 * 0.4 * "x") + "w0d_13_10_5" * COS(5 * 0.4 * "x");
    "phi" := "phi" + "w0c_13_10_6" * SIN(6 * 0.4 * "x") + "w0d_13_10_6" * COS(6 * 0.4 * "x");
    "acc" := "acc" + "phi";
    "x" := "feat_11";
    "phi" := "w0b_13_11" * "x" / (1.0 + EXP(-"x"));
    "phi" := "phi" + "w0c_13_11_1" * SIN(1 * 0.4 * "x") + "w0d_13_11_1" * COS(1 * 0.4 * "x");
    "phi" := "phi" + "w0c_13_11_2" * SIN(2 * 0.4 * "x") + "w0d_13_11_2" * COS(2 * 0.4 * "x");
    "phi" := "phi" + "w0c_13_11_3" * SIN(3 * 0.4 * "x") + "w0d_13_11_3" * COS(3 * 0.4 * "x");
    "phi" := "phi" + "w0c_13_11_4" * SIN(4 * 0.4 * "x") + "w0d_13_11_4" * COS(4 * 0.4 * "x");
    "phi" := "phi" + "w0c_13_11_5" * SIN(5 * 0.4 * "x") + "w0d_13_11_5" * COS(5 * 0.4 * "x");
    "phi" := "phi" + "w0c_13_11_6" * SIN(6 * 0.4 * "x") + "w0d_13_11_6" * COS(6 * 0.4 * "x");
    "acc" := "acc" + "phi";
    "x" := "feat_12";
    "phi" := "w0b_13_12" * "x" / (1.0 + EXP(-"x"));
    "phi" := "phi" + "w0c_13_12_1" * SIN(1 * 0.4 * "x") + "w0d_13_12_1" * COS(1 * 0.4 * "x");
    "phi" := "phi" + "w0c_13_12_2" * SIN(2 * 0.4 * "x") + "w0d_13_12_2" * COS(2 * 0.4 * "x");
    "phi" := "phi" + "w0c_13_12_3" * SIN(3 * 0.4 * "x") + "w0d_13_12_3" * COS(3 * 0.4 * "x");
    "phi" := "phi" + "w0c_13_12_4" * SIN(4 * 0.4 * "x") + "w0d_13_12_4" * COS(4 * 0.4 * "x");
    "phi" := "phi" + "w0c_13_12_5" * SIN(5 * 0.4 * "x") + "w0d_13_12_5" * COS(5 * 0.4 * "x");
    "phi" := "phi" + "w0c_13_12_6" * SIN(6 * 0.4 * "x") + "w0d_13_12_6" * COS(6 * 0.4 * "x");
    "acc" := "acc" + "phi";
    "x" := "feat_13";
    "phi" := "w0b_13_13" * "x" / (1.0 + EXP(-"x"));
    "phi" := "phi" + "w0c_13_13_1" * SIN(1 * 0.4 * "x") + "w0d_13_13_1" * COS(1 * 0.4 * "x");
    "phi" := "phi" + "w0c_13_13_2" * SIN(2 * 0.4 * "x") + "w0d_13_13_2" * COS(2 * 0.4 * "x");
    "phi" := "phi" + "w0c_13_13_3" * SIN(3 * 0.4 * "x") + "w0d_13_13_3" * COS(3 * 0.4 * "x");
    "phi" := "phi" + "w0c_13_13_4" * SIN(4 * 0.4 * "x") + "w0d_13_13_4" * COS(4 * 0.4 * "x");
    "phi" := "phi" + "w0c_13_13_5" * SIN(5 * 0.4 * "x") + "w0d_13_13_5" * COS(5 * 0.4 * "x");
    "phi" := "phi" + "w0c_13_13_6" * SIN(6 * 0.4 * "x") + "w0d_13_13_6" * COS(6 * 0.4 * "x");
    "acc" := "acc" + "phi";
    "x" := "feat_14";
    "phi" := "w0b_13_14" * "x" / (1.0 + EXP(-"x"));
    "phi" := "phi" + "w0c_13_14_1" * SIN(1 * 0.4 * "x") + "w0d_13_14_1" * COS(1 * 0.4 * "x");
    "phi" := "phi" + "w0c_13_14_2" * SIN(2 * 0.4 * "x") + "w0d_13_14_2" * COS(2 * 0.4 * "x");
    "phi" := "phi" + "w0c_13_14_3" * SIN(3 * 0.4 * "x") + "w0d_13_14_3" * COS(3 * 0.4 * "x");
    "phi" := "phi" + "w0c_13_14_4" * SIN(4 * 0.4 * "x") + "w0d_13_14_4" * COS(4 * 0.4 * "x");
    "phi" := "phi" + "w0c_13_14_5" * SIN(5 * 0.4 * "x") + "w0d_13_14_5" * COS(5 * 0.4 * "x");
    "phi" := "phi" + "w0c_13_14_6" * SIN(6 * 0.4 * "x") + "w0d_13_14_6" * COS(6 * 0.4 * "x");
    "acc" := "acc" + "phi";
    "x" := "feat_15";
    "phi" := "w0b_13_15" * "x" / (1.0 + EXP(-"x"));
    "phi" := "phi" + "w0c_13_15_1" * SIN(1 * 0.4 * "x") + "w0d_13_15_1" * COS(1 * 0.4 * "x");
    "phi" := "phi" + "w0c_13_15_2" * SIN(2 * 0.4 * "x") + "w0d_13_15_2" * COS(2 * 0.4 * "x");
    "phi" := "phi" + "w0c_13_15_3" * SIN(3 * 0.4 * "x") + "w0d_13_15_3" * COS(3 * 0.4 * "x");
    "phi" := "phi" + "w0c_13_15_4" * SIN(4 * 0.4 * "x") + "w0d_13_15_4" * COS(4 * 0.4 * "x");
    "phi" := "phi" + "w0c_13_15_5" * SIN(5 * 0.4 * "x") + "w0d_13_15_5" * COS(5 * 0.4 * "x");
    "phi" := "phi" + "w0c_13_15_6" * SIN(6 * 0.4 * "x") + "w0d_13_15_6" * COS(6 * 0.4 * "x");
    "acc" := "acc" + "phi";
    "x" := "feat_16";
    "phi" := "w0b_13_16" * "x" / (1.0 + EXP(-"x"));
    "phi" := "phi" + "w0c_13_16_1" * SIN(1 * 0.4 * "x") + "w0d_13_16_1" * COS(1 * 0.4 * "x");
    "phi" := "phi" + "w0c_13_16_2" * SIN(2 * 0.4 * "x") + "w0d_13_16_2" * COS(2 * 0.4 * "x");
    "phi" := "phi" + "w0c_13_16_3" * SIN(3 * 0.4 * "x") + "w0d_13_16_3" * COS(3 * 0.4 * "x");
    "phi" := "phi" + "w0c_13_16_4" * SIN(4 * 0.4 * "x") + "w0d_13_16_4" * COS(4 * 0.4 * "x");
    "phi" := "phi" + "w0c_13_16_5" * SIN(5 * 0.4 * "x") + "w0d_13_16_5" * COS(5 * 0.4 * "x");
    "phi" := "phi" + "w0c_13_16_6" * SIN(6 * 0.4 * "x") + "w0d_13_16_6" * COS(6 * 0.4 * "x");
    "acc" := "acc" + "phi";
    "x" := "feat_17";
    "phi" := "w0b_13_17" * "x" / (1.0 + EXP(-"x"));
    "phi" := "phi" + "w0c_13_17_1" * SIN(1 * 0.4 * "x") + "w0d_13_17_1" * COS(1 * 0.4 * "x");
    "phi" := "phi" + "w0c_13_17_2" * SIN(2 * 0.4 * "x") + "w0d_13_17_2" * COS(2 * 0.4 * "x");
    "phi" := "phi" + "w0c_13_17_3" * SIN(3 * 0.4 * "x") + "w0d_13_17_3" * COS(3 * 0.4 * "x");
    "phi" := "phi" + "w0c_13_17_4" * SIN(4 * 0.4 * "x") + "w0d_13_17_4" * COS(4 * 0.4 * "x");
    "phi" := "phi" + "w0c_13_17_5" * SIN(5 * 0.4 * "x") + "w0d_13_17_5" * COS(5 * 0.4 * "x");
    "phi" := "phi" + "w0c_13_17_6" * SIN(6 * 0.4 * "x") + "w0d_13_17_6" * COS(6 * 0.4 * "x");
    "acc" := "acc" + "phi";
    "x" := "feat_18";
    "phi" := "w0b_13_18" * "x" / (1.0 + EXP(-"x"));
    "phi" := "phi" + "w0c_13_18_1" * SIN(1 * 0.4 * "x") + "w0d_13_18_1" * COS(1 * 0.4 * "x");
    "phi" := "phi" + "w0c_13_18_2" * SIN(2 * 0.4 * "x") + "w0d_13_18_2" * COS(2 * 0.4 * "x");
    "phi" := "phi" + "w0c_13_18_3" * SIN(3 * 0.4 * "x") + "w0d_13_18_3" * COS(3 * 0.4 * "x");
    "phi" := "phi" + "w0c_13_18_4" * SIN(4 * 0.4 * "x") + "w0d_13_18_4" * COS(4 * 0.4 * "x");
    "phi" := "phi" + "w0c_13_18_5" * SIN(5 * 0.4 * "x") + "w0d_13_18_5" * COS(5 * 0.4 * "x");
    "phi" := "phi" + "w0c_13_18_6" * SIN(6 * 0.4 * "x") + "w0d_13_18_6" * COS(6 * 0.4 * "x");
    "acc" := "acc" + "phi";
    "x" := "feat_19";
    "phi" := "w0b_13_19" * "x" / (1.0 + EXP(-"x"));
    "phi" := "phi" + "w0c_13_19_1" * SIN(1 * 0.4 * "x") + "w0d_13_19_1" * COS(1 * 0.4 * "x");
    "phi" := "phi" + "w0c_13_19_2" * SIN(2 * 0.4 * "x") + "w0d_13_19_2" * COS(2 * 0.4 * "x");
    "phi" := "phi" + "w0c_13_19_3" * SIN(3 * 0.4 * "x") + "w0d_13_19_3" * COS(3 * 0.4 * "x");
    "phi" := "phi" + "w0c_13_19_4" * SIN(4 * 0.4 * "x") + "w0d_13_19_4" * COS(4 * 0.4 * "x");
    "phi" := "phi" + "w0c_13_19_5" * SIN(5 * 0.4 * "x") + "w0d_13_19_5" * COS(5 * 0.4 * "x");
    "phi" := "phi" + "w0c_13_19_6" * SIN(6 * 0.4 * "x") + "w0d_13_19_6" * COS(6 * 0.4 * "x");
    "acc" := "acc" + "phi";
    "x" := "feat_20";
    "phi" := "w0b_13_20" * "x" / (1.0 + EXP(-"x"));
    "phi" := "phi" + "w0c_13_20_1" * SIN(1 * 0.4 * "x") + "w0d_13_20_1" * COS(1 * 0.4 * "x");
    "phi" := "phi" + "w0c_13_20_2" * SIN(2 * 0.4 * "x") + "w0d_13_20_2" * COS(2 * 0.4 * "x");
    "phi" := "phi" + "w0c_13_20_3" * SIN(3 * 0.4 * "x") + "w0d_13_20_3" * COS(3 * 0.4 * "x");
    "phi" := "phi" + "w0c_13_20_4" * SIN(4 * 0.4 * "x") + "w0d_13_20_4" * COS(4 * 0.4 * "x");
    "phi" := "phi" + "w0c_13_20_5" * SIN(5 * 0.4 * "x") + "w0d_13_20_5" * COS(5 * 0.4 * "x");
    "phi" := "phi" + "w0c_13_20_6" * SIN(6 * 0.4 * "x") + "w0d_13_20_6" * COS(6 * 0.4 * "x");
    "acc" := "acc" + "phi";
    "x" := "feat_21";
    "phi" := "w0b_13_21" * "x" / (1.0 + EXP(-"x"));
    "phi" := "phi" + "w0c_13_21_1" * SIN(1 * 0.4 * "x") + "w0d_13_21_1" * COS(1 * 0.4 * "x");
    "phi" := "phi" + "w0c_13_21_2" * SIN(2 * 0.4 * "x") + "w0d_13_21_2" * COS(2 * 0.4 * "x");
    "phi" := "phi" + "w0c_13_21_3" * SIN(3 * 0.4 * "x") + "w0d_13_21_3" * COS(3 * 0.4 * "x");
    "phi" := "phi" + "w0c_13_21_4" * SIN(4 * 0.4 * "x") + "w0d_13_21_4" * COS(4 * 0.4 * "x");
    "phi" := "phi" + "w0c_13_21_5" * SIN(5 * 0.4 * "x") + "w0d_13_21_5" * COS(5 * 0.4 * "x");
    "phi" := "phi" + "w0c_13_21_6" * SIN(6 * 0.4 * "x") + "w0d_13_21_6" * COS(6 * 0.4 * "x");
    "acc" := "acc" + "phi";
    "x" := "feat_22";
    "phi" := "w0b_13_22" * "x" / (1.0 + EXP(-"x"));
    "phi" := "phi" + "w0c_13_22_1" * SIN(1 * 0.4 * "x") + "w0d_13_22_1" * COS(1 * 0.4 * "x");
    "phi" := "phi" + "w0c_13_22_2" * SIN(2 * 0.4 * "x") + "w0d_13_22_2" * COS(2 * 0.4 * "x");
    "phi" := "phi" + "w0c_13_22_3" * SIN(3 * 0.4 * "x") + "w0d_13_22_3" * COS(3 * 0.4 * "x");
    "phi" := "phi" + "w0c_13_22_4" * SIN(4 * 0.4 * "x") + "w0d_13_22_4" * COS(4 * 0.4 * "x");
    "phi" := "phi" + "w0c_13_22_5" * SIN(5 * 0.4 * "x") + "w0d_13_22_5" * COS(5 * 0.4 * "x");
    "phi" := "phi" + "w0c_13_22_6" * SIN(6 * 0.4 * "x") + "w0d_13_22_6" * COS(6 * 0.4 * "x");
    "acc" := "acc" + "phi";
    "x" := "feat_23";
    "phi" := "w0b_13_23" * "x" / (1.0 + EXP(-"x"));
    "phi" := "phi" + "w0c_13_23_1" * SIN(1 * 0.4 * "x") + "w0d_13_23_1" * COS(1 * 0.4 * "x");
    "phi" := "phi" + "w0c_13_23_2" * SIN(2 * 0.4 * "x") + "w0d_13_23_2" * COS(2 * 0.4 * "x");
    "phi" := "phi" + "w0c_13_23_3" * SIN(3 * 0.4 * "x") + "w0d_13_23_3" * COS(3 * 0.4 * "x");
    "phi" := "phi" + "w0c_13_23_4" * SIN(4 * 0.4 * "x") + "w0d_13_23_4" * COS(4 * 0.4 * "x");
    "phi" := "phi" + "w0c_13_23_5" * SIN(5 * 0.4 * "x") + "w0d_13_23_5" * COS(5 * 0.4 * "x");
    "phi" := "phi" + "w0c_13_23_6" * SIN(6 * 0.4 * "x") + "w0d_13_23_6" * COS(6 * 0.4 * "x");
    "acc" := "acc" + "phi";
    "x" := "feat_24";
    "phi" := "w0b_13_24" * "x" / (1.0 + EXP(-"x"));
    "phi" := "phi" + "w0c_13_24_1" * SIN(1 * 0.4 * "x") + "w0d_13_24_1" * COS(1 * 0.4 * "x");
    "phi" := "phi" + "w0c_13_24_2" * SIN(2 * 0.4 * "x") + "w0d_13_24_2" * COS(2 * 0.4 * "x");
    "phi" := "phi" + "w0c_13_24_3" * SIN(3 * 0.4 * "x") + "w0d_13_24_3" * COS(3 * 0.4 * "x");
    "phi" := "phi" + "w0c_13_24_4" * SIN(4 * 0.4 * "x") + "w0d_13_24_4" * COS(4 * 0.4 * "x");
    "phi" := "phi" + "w0c_13_24_5" * SIN(5 * 0.4 * "x") + "w0d_13_24_5" * COS(5 * 0.4 * "x");
    "phi" := "phi" + "w0c_13_24_6" * SIN(6 * 0.4 * "x") + "w0d_13_24_6" * COS(6 * 0.4 * "x");
    "acc" := "acc" + "phi";
    "x" := "feat_25";
    "phi" := "w0b_13_25" * "x" / (1.0 + EXP(-"x"));
    "phi" := "phi" + "w0c_13_25_1" * SIN(1 * 0.4 * "x") + "w0d_13_25_1" * COS(1 * 0.4 * "x");
    "phi" := "phi" + "w0c_13_25_2" * SIN(2 * 0.4 * "x") + "w0d_13_25_2" * COS(2 * 0.4 * "x");
    "phi" := "phi" + "w0c_13_25_3" * SIN(3 * 0.4 * "x") + "w0d_13_25_3" * COS(3 * 0.4 * "x");
    "phi" := "phi" + "w0c_13_25_4" * SIN(4 * 0.4 * "x") + "w0d_13_25_4" * COS(4 * 0.4 * "x");
    "phi" := "phi" + "w0c_13_25_5" * SIN(5 * 0.4 * "x") + "w0d_13_25_5" * COS(5 * 0.4 * "x");
    "phi" := "phi" + "w0c_13_25_6" * SIN(6 * 0.4 * "x") + "w0d_13_25_6" * COS(6 * 0.4 * "x");
    "acc" := "acc" + "phi";
    "x" := "feat_26";
    "phi" := "w0b_13_26" * "x" / (1.0 + EXP(-"x"));
    "phi" := "phi" + "w0c_13_26_1" * SIN(1 * 0.4 * "x") + "w0d_13_26_1" * COS(1 * 0.4 * "x");
    "phi" := "phi" + "w0c_13_26_2" * SIN(2 * 0.4 * "x") + "w0d_13_26_2" * COS(2 * 0.4 * "x");
    "phi" := "phi" + "w0c_13_26_3" * SIN(3 * 0.4 * "x") + "w0d_13_26_3" * COS(3 * 0.4 * "x");
    "phi" := "phi" + "w0c_13_26_4" * SIN(4 * 0.4 * "x") + "w0d_13_26_4" * COS(4 * 0.4 * "x");
    "phi" := "phi" + "w0c_13_26_5" * SIN(5 * 0.4 * "x") + "w0d_13_26_5" * COS(5 * 0.4 * "x");
    "phi" := "phi" + "w0c_13_26_6" * SIN(6 * 0.4 * "x") + "w0d_13_26_6" * COS(6 * 0.4 * "x");
    "acc" := "acc" + "phi";
    "x" := "feat_27";
    "phi" := "w0b_13_27" * "x" / (1.0 + EXP(-"x"));
    "phi" := "phi" + "w0c_13_27_1" * SIN(1 * 0.4 * "x") + "w0d_13_27_1" * COS(1 * 0.4 * "x");
    "phi" := "phi" + "w0c_13_27_2" * SIN(2 * 0.4 * "x") + "w0d_13_27_2" * COS(2 * 0.4 * "x");
    "phi" := "phi" + "w0c_13_27_3" * SIN(3 * 0.4 * "x") + "w0d_13_27_3" * COS(3 * 0.4 * "x");
    "phi" := "phi" + "w0c_13_27_4" * SIN(4 * 0.4 * "x") + "w0d_13_27_4" * COS(4 * 0.4 * "x");
    "phi" := "phi" + "w0c_13_27_5" * SIN(5 * 0.4 * "x") + "w0d_13_27_5" * COS(5 * 0.4 * "x");
    "phi" := "phi" + "w0c_13_27_6" * SIN(6 * 0.4 * "x") + "w0d_13_27_6" * COS(6 * 0.4 * "x");
    "acc" := "acc" + "phi";
    "x" := "feat_28";
    "phi" := "w0b_13_28" * "x" / (1.0 + EXP(-"x"));
    "phi" := "phi" + "w0c_13_28_1" * SIN(1 * 0.4 * "x") + "w0d_13_28_1" * COS(1 * 0.4 * "x");
    "phi" := "phi" + "w0c_13_28_2" * SIN(2 * 0.4 * "x") + "w0d_13_28_2" * COS(2 * 0.4 * "x");
    "phi" := "phi" + "w0c_13_28_3" * SIN(3 * 0.4 * "x") + "w0d_13_28_3" * COS(3 * 0.4 * "x");
    "phi" := "phi" + "w0c_13_28_4" * SIN(4 * 0.4 * "x") + "w0d_13_28_4" * COS(4 * 0.4 * "x");
    "phi" := "phi" + "w0c_13_28_5" * SIN(5 * 0.4 * "x") + "w0d_13_28_5" * COS(5 * 0.4 * "x");
    "phi" := "phi" + "w0c_13_28_6" * SIN(6 * 0.4 * "x") + "w0d_13_28_6" * COS(6 * 0.4 * "x");
    "acc" := "acc" + "phi";
    "h1_13" := "acc" + "b0_13";
    "acc" := 0.0;
    "x" := "feat_1";
    "phi" := "w0b_14_1" * "x" / (1.0 + EXP(-"x"));
    "phi" := "phi" + "w0c_14_1_1" * SIN(1 * 0.4 * "x") + "w0d_14_1_1" * COS(1 * 0.4 * "x");
    "phi" := "phi" + "w0c_14_1_2" * SIN(2 * 0.4 * "x") + "w0d_14_1_2" * COS(2 * 0.4 * "x");
    "phi" := "phi" + "w0c_14_1_3" * SIN(3 * 0.4 * "x") + "w0d_14_1_3" * COS(3 * 0.4 * "x");
    "phi" := "phi" + "w0c_14_1_4" * SIN(4 * 0.4 * "x") + "w0d_14_1_4" * COS(4 * 0.4 * "x");
    "phi" := "phi" + "w0c_14_1_5" * SIN(5 * 0.4 * "x") + "w0d_14_1_5" * COS(5 * 0.4 * "x");
    "phi" := "phi" + "w0c_14_1_6" * SIN(6 * 0.4 * "x") + "w0d_14_1_6" * COS(6 * 0.4 * "x");
    "acc" := "acc" + "phi";
    "x" := "feat_2";
    "phi" := "w0b_14_2" * "x" / (1.0 + EXP(-"x"));
    "phi" := "phi" + "w0c_14_2_1" * SIN(1 * 0.4 * "x") + "w0d_14_2_1" * COS(1 * 0.4 * "x");
    "phi" := "phi" + "w0c_14_2_2" * SIN(2 * 0.4 * "x") + "w0d_14_2_2" * COS(2 * 0.4 * "x");
    "phi" := "phi" + "w0c_14_2_3" * SIN(3 * 0.4 * "x") + "w0d_14_2_3" * COS(3 * 0.4 * "x");
    "phi" := "phi" + "w0c_14_2_4" * SIN(4 * 0.4 * "x") + "w0d_14_2_4" * COS(4 * 0.4 * "x");
    "phi" := "phi" + "w0c_14_2_5" * SIN(5 * 0.4 * "x") + "w0d_14_2_5" * COS(5 * 0.4 * "x");
    "phi" := "phi" + "w0c_14_2_6" * SIN(6 * 0.4 * "x") + "w0d_14_2_6" * COS(6 * 0.4 * "x");
    "acc" := "acc" + "phi";
    "x" := "feat_3";
    "phi" := "w0b_14_3" * "x" / (1.0 + EXP(-"x"));
    "phi" := "phi" + "w0c_14_3_1" * SIN(1 * 0.4 * "x") + "w0d_14_3_1" * COS(1 * 0.4 * "x");
    "phi" := "phi" + "w0c_14_3_2" * SIN(2 * 0.4 * "x") + "w0d_14_3_2" * COS(2 * 0.4 * "x");
    "phi" := "phi" + "w0c_14_3_3" * SIN(3 * 0.4 * "x") + "w0d_14_3_3" * COS(3 * 0.4 * "x");
    "phi" := "phi" + "w0c_14_3_4" * SIN(4 * 0.4 * "x") + "w0d_14_3_4" * COS(4 * 0.4 * "x");
    "phi" := "phi" + "w0c_14_3_5" * SIN(5 * 0.4 * "x") + "w0d_14_3_5" * COS(5 * 0.4 * "x");
    "phi" := "phi" + "w0c_14_3_6" * SIN(6 * 0.4 * "x") + "w0d_14_3_6" * COS(6 * 0.4 * "x");
    "acc" := "acc" + "phi";
    "x" := "feat_4";
    "phi" := "w0b_14_4" * "x" / (1.0 + EXP(-"x"));
    "phi" := "phi" + "w0c_14_4_1" * SIN(1 * 0.4 * "x") + "w0d_14_4_1" * COS(1 * 0.4 * "x");
    "phi" := "phi" + "w0c_14_4_2" * SIN(2 * 0.4 * "x") + "w0d_14_4_2" * COS(2 * 0.4 * "x");
    "phi" := "phi" + "w0c_14_4_3" * SIN(3 * 0.4 * "x") + "w0d_14_4_3" * COS(3 * 0.4 * "x");
    "phi" := "phi" + "w0c_14_4_4" * SIN(4 * 0.4 * "x") + "w0d_14_4_4" * COS(4 * 0.4 * "x");
    "phi" := "phi" + "w0c_14_4_5" * SIN(5 * 0.4 * "x") + "w0d_14_4_5" * COS(5 * 0.4 * "x");
    "phi" := "phi" + "w0c_14_4_6" * SIN(6 * 0.4 * "x") + "w0d_14_4_6" * COS(6 * 0.4 * "x");
    "acc" := "acc" + "phi";
    "x" := "feat_5";
    "phi" := "w0b_14_5" * "x" / (1.0 + EXP(-"x"));
    "phi" := "phi" + "w0c_14_5_1" * SIN(1 * 0.4 * "x") + "w0d_14_5_1" * COS(1 * 0.4 * "x");
    "phi" := "phi" + "w0c_14_5_2" * SIN(2 * 0.4 * "x") + "w0d_14_5_2" * COS(2 * 0.4 * "x");
    "phi" := "phi" + "w0c_14_5_3" * SIN(3 * 0.4 * "x") + "w0d_14_5_3" * COS(3 * 0.4 * "x");
    "phi" := "phi" + "w0c_14_5_4" * SIN(4 * 0.4 * "x") + "w0d_14_5_4" * COS(4 * 0.4 * "x");
    "phi" := "phi" + "w0c_14_5_5" * SIN(5 * 0.4 * "x") + "w0d_14_5_5" * COS(5 * 0.4 * "x");
    "phi" := "phi" + "w0c_14_5_6" * SIN(6 * 0.4 * "x") + "w0d_14_5_6" * COS(6 * 0.4 * "x");
    "acc" := "acc" + "phi";
    "x" := "feat_6";
    "phi" := "w0b_14_6" * "x" / (1.0 + EXP(-"x"));
    "phi" := "phi" + "w0c_14_6_1" * SIN(1 * 0.4 * "x") + "w0d_14_6_1" * COS(1 * 0.4 * "x");
    "phi" := "phi" + "w0c_14_6_2" * SIN(2 * 0.4 * "x") + "w0d_14_6_2" * COS(2 * 0.4 * "x");
    "phi" := "phi" + "w0c_14_6_3" * SIN(3 * 0.4 * "x") + "w0d_14_6_3" * COS(3 * 0.4 * "x");
    "phi" := "phi" + "w0c_14_6_4" * SIN(4 * 0.4 * "x") + "w0d_14_6_4" * COS(4 * 0.4 * "x");
    "phi" := "phi" + "w0c_14_6_5" * SIN(5 * 0.4 * "x") + "w0d_14_6_5" * COS(5 * 0.4 * "x");
    "phi" := "phi" + "w0c_14_6_6" * SIN(6 * 0.4 * "x") + "w0d_14_6_6" * COS(6 * 0.4 * "x");
    "acc" := "acc" + "phi";
    "x" := "feat_7";
    "phi" := "w0b_14_7" * "x" / (1.0 + EXP(-"x"));
    "phi" := "phi" + "w0c_14_7_1" * SIN(1 * 0.4 * "x") + "w0d_14_7_1" * COS(1 * 0.4 * "x");
    "phi" := "phi" + "w0c_14_7_2" * SIN(2 * 0.4 * "x") + "w0d_14_7_2" * COS(2 * 0.4 * "x");
    "phi" := "phi" + "w0c_14_7_3" * SIN(3 * 0.4 * "x") + "w0d_14_7_3" * COS(3 * 0.4 * "x");
    "phi" := "phi" + "w0c_14_7_4" * SIN(4 * 0.4 * "x") + "w0d_14_7_4" * COS(4 * 0.4 * "x");
    "phi" := "phi" + "w0c_14_7_5" * SIN(5 * 0.4 * "x") + "w0d_14_7_5" * COS(5 * 0.4 * "x");
    "phi" := "phi" + "w0c_14_7_6" * SIN(6 * 0.4 * "x") + "w0d_14_7_6" * COS(6 * 0.4 * "x");
    "acc" := "acc" + "phi";
    "x" := "feat_8";
    "phi" := "w0b_14_8" * "x" / (1.0 + EXP(-"x"));
    "phi" := "phi" + "w0c_14_8_1" * SIN(1 * 0.4 * "x") + "w0d_14_8_1" * COS(1 * 0.4 * "x");
    "phi" := "phi" + "w0c_14_8_2" * SIN(2 * 0.4 * "x") + "w0d_14_8_2" * COS(2 * 0.4 * "x");
    "phi" := "phi" + "w0c_14_8_3" * SIN(3 * 0.4 * "x") + "w0d_14_8_3" * COS(3 * 0.4 * "x");
    "phi" := "phi" + "w0c_14_8_4" * SIN(4 * 0.4 * "x") + "w0d_14_8_4" * COS(4 * 0.4 * "x");
    "phi" := "phi" + "w0c_14_8_5" * SIN(5 * 0.4 * "x") + "w0d_14_8_5" * COS(5 * 0.4 * "x");
    "phi" := "phi" + "w0c_14_8_6" * SIN(6 * 0.4 * "x") + "w0d_14_8_6" * COS(6 * 0.4 * "x");
    "acc" := "acc" + "phi";
    "x" := "feat_9";
    "phi" := "w0b_14_9" * "x" / (1.0 + EXP(-"x"));
    "phi" := "phi" + "w0c_14_9_1" * SIN(1 * 0.4 * "x") + "w0d_14_9_1" * COS(1 * 0.4 * "x");
    "phi" := "phi" + "w0c_14_9_2" * SIN(2 * 0.4 * "x") + "w0d_14_9_2" * COS(2 * 0.4 * "x");
    "phi" := "phi" + "w0c_14_9_3" * SIN(3 * 0.4 * "x") + "w0d_14_9_3" * COS(3 * 0.4 * "x");
    "phi" := "phi" + "w0c_14_9_4" * SIN(4 * 0.4 * "x") + "w0d_14_9_4" * COS(4 * 0.4 * "x");
    "phi" := "phi" + "w0c_14_9_5" * SIN(5 * 0.4 * "x") + "w0d_14_9_5" * COS(5 * 0.4 * "x");
    "phi" := "phi" + "w0c_14_9_6" * SIN(6 * 0.4 * "x") + "w0d_14_9_6" * COS(6 * 0.4 * "x");
    "acc" := "acc" + "phi";
    "x" := "feat_10";
    "phi" := "w0b_14_10" * "x" / (1.0 + EXP(-"x"));
    "phi" := "phi" + "w0c_14_10_1" * SIN(1 * 0.4 * "x") + "w0d_14_10_1" * COS(1 * 0.4 * "x");
    "phi" := "phi" + "w0c_14_10_2" * SIN(2 * 0.4 * "x") + "w0d_14_10_2" * COS(2 * 0.4 * "x");
    "phi" := "phi" + "w0c_14_10_3" * SIN(3 * 0.4 * "x") + "w0d_14_10_3" * COS(3 * 0.4 * "x");
    "phi" := "phi" + "w0c_14_10_4" * SIN(4 * 0.4 * "x") + "w0d_14_10_4" * COS(4 * 0.4 * "x");
    "phi" := "phi" + "w0c_14_10_5" * SIN(5 * 0.4 * "x") + "w0d_14_10_5" * COS(5 * 0.4 * "x");
    "phi" := "phi" + "w0c_14_10_6" * SIN(6 * 0.4 * "x") + "w0d_14_10_6" * COS(6 * 0.4 * "x");
    "acc" := "acc" + "phi";
    "x" := "feat_11";
    "phi" := "w0b_14_11" * "x" / (1.0 + EXP(-"x"));
    "phi" := "phi" + "w0c_14_11_1" * SIN(1 * 0.4 * "x") + "w0d_14_11_1" * COS(1 * 0.4 * "x");
    "phi" := "phi" + "w0c_14_11_2" * SIN(2 * 0.4 * "x") + "w0d_14_11_2" * COS(2 * 0.4 * "x");
    "phi" := "phi" + "w0c_14_11_3" * SIN(3 * 0.4 * "x") + "w0d_14_11_3" * COS(3 * 0.4 * "x");
    "phi" := "phi" + "w0c_14_11_4" * SIN(4 * 0.4 * "x") + "w0d_14_11_4" * COS(4 * 0.4 * "x");
    "phi" := "phi" + "w0c_14_11_5" * SIN(5 * 0.4 * "x") + "w0d_14_11_5" * COS(5 * 0.4 * "x");
    "phi" := "phi" + "w0c_14_11_6" * SIN(6 * 0.4 * "x") + "w0d_14_11_6" * COS(6 * 0.4 * "x");
    "acc" := "acc" + "phi";
    "x" := "feat_12";
    "phi" := "w0b_14_12" * "x" / (1.0 + EXP(-"x"));
    "phi" := "phi" + "w0c_14_12_1" * SIN(1 * 0.4 * "x") + "w0d_14_12_1" * COS(1 * 0.4 * "x");
    "phi" := "phi" + "w0c_14_12_2" * SIN(2 * 0.4 * "x") + "w0d_14_12_2" * COS(2 * 0.4 * "x");
    "phi" := "phi" + "w0c_14_12_3" * SIN(3 * 0.4 * "x") + "w0d_14_12_3" * COS(3 * 0.4 * "x");
    "phi" := "phi" + "w0c_14_12_4" * SIN(4 * 0.4 * "x") + "w0d_14_12_4" * COS(4 * 0.4 * "x");
    "phi" := "phi" + "w0c_14_12_5" * SIN(5 * 0.4 * "x") + "w0d_14_12_5" * COS(5 * 0.4 * "x");
    "phi" := "phi" + "w0c_14_12_6" * SIN(6 * 0.4 * "x") + "w0d_14_12_6" * COS(6 * 0.4 * "x");
    "acc" := "acc" + "phi";
    "x" := "feat_13";
    "phi" := "w0b_14_13" * "x" / (1.0 + EXP(-"x"));
    "phi" := "phi" + "w0c_14_13_1" * SIN(1 * 0.4 * "x") + "w0d_14_13_1" * COS(1 * 0.4 * "x");
    "phi" := "phi" + "w0c_14_13_2" * SIN(2 * 0.4 * "x") + "w0d_14_13_2" * COS(2 * 0.4 * "x");
    "phi" := "phi" + "w0c_14_13_3" * SIN(3 * 0.4 * "x") + "w0d_14_13_3" * COS(3 * 0.4 * "x");
    "phi" := "phi" + "w0c_14_13_4" * SIN(4 * 0.4 * "x") + "w0d_14_13_4" * COS(4 * 0.4 * "x");
    "phi" := "phi" + "w0c_14_13_5" * SIN(5 * 0.4 * "x") + "w0d_14_13_5" * COS(5 * 0.4 * "x");
    "phi" := "phi" + "w0c_14_13_6" * SIN(6 * 0.4 * "x") + "w0d_14_13_6" * COS(6 * 0.4 * "x");
    "acc" := "acc" + "phi";
    "x" := "feat_14";
    "phi" := "w0b_14_14" * "x" / (1.0 + EXP(-"x"));
    "phi" := "phi" + "w0c_14_14_1" * SIN(1 * 0.4 * "x") + "w0d_14_14_1" * COS(1 * 0.4 * "x");
    "phi" := "phi" + "w0c_14_14_2" * SIN(2 * 0.4 * "x") + "w0d_14_14_2" * COS(2 * 0.4 * "x");
    "phi" := "phi" + "w0c_14_14_3" * SIN(3 * 0.4 * "x") + "w0d_14_14_3" * COS(3 * 0.4 * "x");
    "phi" := "phi" + "w0c_14_14_4" * SIN(4 * 0.4 * "x") + "w0d_14_14_4" * COS(4 * 0.4 * "x");
    "phi" := "phi" + "w0c_14_14_5" * SIN(5 * 0.4 * "x") + "w0d_14_14_5" * COS(5 * 0.4 * "x");
    "phi" := "phi" + "w0c_14_14_6" * SIN(6 * 0.4 * "x") + "w0d_14_14_6" * COS(6 * 0.4 * "x");
    "acc" := "acc" + "phi";
    "x" := "feat_15";
    "phi" := "w0b_14_15" * "x" / (1.0 + EXP(-"x"));
    "phi" := "phi" + "w0c_14_15_1" * SIN(1 * 0.4 * "x") + "w0d_14_15_1" * COS(1 * 0.4 * "x");
    "phi" := "phi" + "w0c_14_15_2" * SIN(2 * 0.4 * "x") + "w0d_14_15_2" * COS(2 * 0.4 * "x");
    "phi" := "phi" + "w0c_14_15_3" * SIN(3 * 0.4 * "x") + "w0d_14_15_3" * COS(3 * 0.4 * "x");
    "phi" := "phi" + "w0c_14_15_4" * SIN(4 * 0.4 * "x") + "w0d_14_15_4" * COS(4 * 0.4 * "x");
    "phi" := "phi" + "w0c_14_15_5" * SIN(5 * 0.4 * "x") + "w0d_14_15_5" * COS(5 * 0.4 * "x");
    "phi" := "phi" + "w0c_14_15_6" * SIN(6 * 0.4 * "x") + "w0d_14_15_6" * COS(6 * 0.4 * "x");
    "acc" := "acc" + "phi";
    "x" := "feat_16";
    "phi" := "w0b_14_16" * "x" / (1.0 + EXP(-"x"));
    "phi" := "phi" + "w0c_14_16_1" * SIN(1 * 0.4 * "x") + "w0d_14_16_1" * COS(1 * 0.4 * "x");
    "phi" := "phi" + "w0c_14_16_2" * SIN(2 * 0.4 * "x") + "w0d_14_16_2" * COS(2 * 0.4 * "x");
    "phi" := "phi" + "w0c_14_16_3" * SIN(3 * 0.4 * "x") + "w0d_14_16_3" * COS(3 * 0.4 * "x");
    "phi" := "phi" + "w0c_14_16_4" * SIN(4 * 0.4 * "x") + "w0d_14_16_4" * COS(4 * 0.4 * "x");
    "phi" := "phi" + "w0c_14_16_5" * SIN(5 * 0.4 * "x") + "w0d_14_16_5" * COS(5 * 0.4 * "x");
    "phi" := "phi" + "w0c_14_16_6" * SIN(6 * 0.4 * "x") + "w0d_14_16_6" * COS(6 * 0.4 * "x");
    "acc" := "acc" + "phi";
    "x" := "feat_17";
    "phi" := "w0b_14_17" * "x" / (1.0 + EXP(-"x"));
    "phi" := "phi" + "w0c_14_17_1" * SIN(1 * 0.4 * "x") + "w0d_14_17_1" * COS(1 * 0.4 * "x");
    "phi" := "phi" + "w0c_14_17_2" * SIN(2 * 0.4 * "x") + "w0d_14_17_2" * COS(2 * 0.4 * "x");
    "phi" := "phi" + "w0c_14_17_3" * SIN(3 * 0.4 * "x") + "w0d_14_17_3" * COS(3 * 0.4 * "x");
    "phi" := "phi" + "w0c_14_17_4" * SIN(4 * 0.4 * "x") + "w0d_14_17_4" * COS(4 * 0.4 * "x");
    "phi" := "phi" + "w0c_14_17_5" * SIN(5 * 0.4 * "x") + "w0d_14_17_5" * COS(5 * 0.4 * "x");
    "phi" := "phi" + "w0c_14_17_6" * SIN(6 * 0.4 * "x") + "w0d_14_17_6" * COS(6 * 0.4 * "x");
    "acc" := "acc" + "phi";
    "x" := "feat_18";
    "phi" := "w0b_14_18" * "x" / (1.0 + EXP(-"x"));
    "phi" := "phi" + "w0c_14_18_1" * SIN(1 * 0.4 * "x") + "w0d_14_18_1" * COS(1 * 0.4 * "x");
    "phi" := "phi" + "w0c_14_18_2" * SIN(2 * 0.4 * "x") + "w0d_14_18_2" * COS(2 * 0.4 * "x");
    "phi" := "phi" + "w0c_14_18_3" * SIN(3 * 0.4 * "x") + "w0d_14_18_3" * COS(3 * 0.4 * "x");
    "phi" := "phi" + "w0c_14_18_4" * SIN(4 * 0.4 * "x") + "w0d_14_18_4" * COS(4 * 0.4 * "x");
    "phi" := "phi" + "w0c_14_18_5" * SIN(5 * 0.4 * "x") + "w0d_14_18_5" * COS(5 * 0.4 * "x");
    "phi" := "phi" + "w0c_14_18_6" * SIN(6 * 0.4 * "x") + "w0d_14_18_6" * COS(6 * 0.4 * "x");
    "acc" := "acc" + "phi";
    "x" := "feat_19";
    "phi" := "w0b_14_19" * "x" / (1.0 + EXP(-"x"));
    "phi" := "phi" + "w0c_14_19_1" * SIN(1 * 0.4 * "x") + "w0d_14_19_1" * COS(1 * 0.4 * "x");
    "phi" := "phi" + "w0c_14_19_2" * SIN(2 * 0.4 * "x") + "w0d_14_19_2" * COS(2 * 0.4 * "x");
    "phi" := "phi" + "w0c_14_19_3" * SIN(3 * 0.4 * "x") + "w0d_14_19_3" * COS(3 * 0.4 * "x");
    "phi" := "phi" + "w0c_14_19_4" * SIN(4 * 0.4 * "x") + "w0d_14_19_4" * COS(4 * 0.4 * "x");
    "phi" := "phi" + "w0c_14_19_5" * SIN(5 * 0.4 * "x") + "w0d_14_19_5" * COS(5 * 0.4 * "x");
    "phi" := "phi" + "w0c_14_19_6" * SIN(6 * 0.4 * "x") + "w0d_14_19_6" * COS(6 * 0.4 * "x");
    "acc" := "acc" + "phi";
    "x" := "feat_20";
    "phi" := "w0b_14_20" * "x" / (1.0 + EXP(-"x"));
    "phi" := "phi" + "w0c_14_20_1" * SIN(1 * 0.4 * "x") + "w0d_14_20_1" * COS(1 * 0.4 * "x");
    "phi" := "phi" + "w0c_14_20_2" * SIN(2 * 0.4 * "x") + "w0d_14_20_2" * COS(2 * 0.4 * "x");
    "phi" := "phi" + "w0c_14_20_3" * SIN(3 * 0.4 * "x") + "w0d_14_20_3" * COS(3 * 0.4 * "x");
    "phi" := "phi" + "w0c_14_20_4" * SIN(4 * 0.4 * "x") + "w0d_14_20_4" * COS(4 * 0.4 * "x");
    "phi" := "phi" + "w0c_14_20_5" * SIN(5 * 0.4 * "x") + "w0d_14_20_5" * COS(5 * 0.4 * "x");
    "phi" := "phi" + "w0c_14_20_6" * SIN(6 * 0.4 * "x") + "w0d_14_20_6" * COS(6 * 0.4 * "x");
    "acc" := "acc" + "phi";
    "x" := "feat_21";
    "phi" := "w0b_14_21" * "x" / (1.0 + EXP(-"x"));
    "phi" := "phi" + "w0c_14_21_1" * SIN(1 * 0.4 * "x") + "w0d_14_21_1" * COS(1 * 0.4 * "x");
    "phi" := "phi" + "w0c_14_21_2" * SIN(2 * 0.4 * "x") + "w0d_14_21_2" * COS(2 * 0.4 * "x");
    "phi" := "phi" + "w0c_14_21_3" * SIN(3 * 0.4 * "x") + "w0d_14_21_3" * COS(3 * 0.4 * "x");
    "phi" := "phi" + "w0c_14_21_4" * SIN(4 * 0.4 * "x") + "w0d_14_21_4" * COS(4 * 0.4 * "x");
    "phi" := "phi" + "w0c_14_21_5" * SIN(5 * 0.4 * "x") + "w0d_14_21_5" * COS(5 * 0.4 * "x");
    "phi" := "phi" + "w0c_14_21_6" * SIN(6 * 0.4 * "x") + "w0d_14_21_6" * COS(6 * 0.4 * "x");
    "acc" := "acc" + "phi";
    "x" := "feat_22";
    "phi" := "w0b_14_22" * "x" / (1.0 + EXP(-"x"));
    "phi" := "phi" + "w0c_14_22_1" * SIN(1 * 0.4 * "x") + "w0d_14_22_1" * COS(1 * 0.4 * "x");
    "phi" := "phi" + "w0c_14_22_2" * SIN(2 * 0.4 * "x") + "w0d_14_22_2" * COS(2 * 0.4 * "x");
    "phi" := "phi" + "w0c_14_22_3" * SIN(3 * 0.4 * "x") + "w0d_14_22_3" * COS(3 * 0.4 * "x");
    "phi" := "phi" + "w0c_14_22_4" * SIN(4 * 0.4 * "x") + "w0d_14_22_4" * COS(4 * 0.4 * "x");
    "phi" := "phi" + "w0c_14_22_5" * SIN(5 * 0.4 * "x") + "w0d_14_22_5" * COS(5 * 0.4 * "x");
    "phi" := "phi" + "w0c_14_22_6" * SIN(6 * 0.4 * "x") + "w0d_14_22_6" * COS(6 * 0.4 * "x");
    "acc" := "acc" + "phi";
    "x" := "feat_23";
    "phi" := "w0b_14_23" * "x" / (1.0 + EXP(-"x"));
    "phi" := "phi" + "w0c_14_23_1" * SIN(1 * 0.4 * "x") + "w0d_14_23_1" * COS(1 * 0.4 * "x");
    "phi" := "phi" + "w0c_14_23_2" * SIN(2 * 0.4 * "x") + "w0d_14_23_2" * COS(2 * 0.4 * "x");
    "phi" := "phi" + "w0c_14_23_3" * SIN(3 * 0.4 * "x") + "w0d_14_23_3" * COS(3 * 0.4 * "x");
    "phi" := "phi" + "w0c_14_23_4" * SIN(4 * 0.4 * "x") + "w0d_14_23_4" * COS(4 * 0.4 * "x");
    "phi" := "phi" + "w0c_14_23_5" * SIN(5 * 0.4 * "x") + "w0d_14_23_5" * COS(5 * 0.4 * "x");
    "phi" := "phi" + "w0c_14_23_6" * SIN(6 * 0.4 * "x") + "w0d_14_23_6" * COS(6 * 0.4 * "x");
    "acc" := "acc" + "phi";
    "x" := "feat_24";
    "phi" := "w0b_14_24" * "x" / (1.0 + EXP(-"x"));
    "phi" := "phi" + "w0c_14_24_1" * SIN(1 * 0.4 * "x") + "w0d_14_24_1" * COS(1 * 0.4 * "x");
    "phi" := "phi" + "w0c_14_24_2" * SIN(2 * 0.4 * "x") + "w0d_14_24_2" * COS(2 * 0.4 * "x");
    "phi" := "phi" + "w0c_14_24_3" * SIN(3 * 0.4 * "x") + "w0d_14_24_3" * COS(3 * 0.4 * "x");
    "phi" := "phi" + "w0c_14_24_4" * SIN(4 * 0.4 * "x") + "w0d_14_24_4" * COS(4 * 0.4 * "x");
    "phi" := "phi" + "w0c_14_24_5" * SIN(5 * 0.4 * "x") + "w0d_14_24_5" * COS(5 * 0.4 * "x");
    "phi" := "phi" + "w0c_14_24_6" * SIN(6 * 0.4 * "x") + "w0d_14_24_6" * COS(6 * 0.4 * "x");
    "acc" := "acc" + "phi";
    "x" := "feat_25";
    "phi" := "w0b_14_25" * "x" / (1.0 + EXP(-"x"));
    "phi" := "phi" + "w0c_14_25_1" * SIN(1 * 0.4 * "x") + "w0d_14_25_1" * COS(1 * 0.4 * "x");
    "phi" := "phi" + "w0c_14_25_2" * SIN(2 * 0.4 * "x") + "w0d_14_25_2" * COS(2 * 0.4 * "x");
    "phi" := "phi" + "w0c_14_25_3" * SIN(3 * 0.4 * "x") + "w0d_14_25_3" * COS(3 * 0.4 * "x");
    "phi" := "phi" + "w0c_14_25_4" * SIN(4 * 0.4 * "x") + "w0d_14_25_4" * COS(4 * 0.4 * "x");
    "phi" := "phi" + "w0c_14_25_5" * SIN(5 * 0.4 * "x") + "w0d_14_25_5" * COS(5 * 0.4 * "x");
    "phi" := "phi" + "w0c_14_25_6" * SIN(6 * 0.4 * "x") + "w0d_14_25_6" * COS(6 * 0.4 * "x");
    "acc" := "acc" + "phi";
    "x" := "feat_26";
    "phi" := "w0b_14_26" * "x" / (1.0 + EXP(-"x"));
    "phi" := "phi" + "w0c_14_26_1" * SIN(1 * 0.4 * "x") + "w0d_14_26_1" * COS(1 * 0.4 * "x");
    "phi" := "phi" + "w0c_14_26_2" * SIN(2 * 0.4 * "x") + "w0d_14_26_2" * COS(2 * 0.4 * "x");
    "phi" := "phi" + "w0c_14_26_3" * SIN(3 * 0.4 * "x") + "w0d_14_26_3" * COS(3 * 0.4 * "x");
    "phi" := "phi" + "w0c_14_26_4" * SIN(4 * 0.4 * "x") + "w0d_14_26_4" * COS(4 * 0.4 * "x");
    "phi" := "phi" + "w0c_14_26_5" * SIN(5 * 0.4 * "x") + "w0d_14_26_5" * COS(5 * 0.4 * "x");
    "phi" := "phi" + "w0c_14_26_6" * SIN(6 * 0.4 * "x") + "w0d_14_26_6" * COS(6 * 0.4 * "x");
    "acc" := "acc" + "phi";
    "x" := "feat_27";
    "phi" := "w0b_14_27" * "x" / (1.0 + EXP(-"x"));
    "phi" := "phi" + "w0c_14_27_1" * SIN(1 * 0.4 * "x") + "w0d_14_27_1" * COS(1 * 0.4 * "x");
    "phi" := "phi" + "w0c_14_27_2" * SIN(2 * 0.4 * "x") + "w0d_14_27_2" * COS(2 * 0.4 * "x");
    "phi" := "phi" + "w0c_14_27_3" * SIN(3 * 0.4 * "x") + "w0d_14_27_3" * COS(3 * 0.4 * "x");
    "phi" := "phi" + "w0c_14_27_4" * SIN(4 * 0.4 * "x") + "w0d_14_27_4" * COS(4 * 0.4 * "x");
    "phi" := "phi" + "w0c_14_27_5" * SIN(5 * 0.4 * "x") + "w0d_14_27_5" * COS(5 * 0.4 * "x");
    "phi" := "phi" + "w0c_14_27_6" * SIN(6 * 0.4 * "x") + "w0d_14_27_6" * COS(6 * 0.4 * "x");
    "acc" := "acc" + "phi";
    "x" := "feat_28";
    "phi" := "w0b_14_28" * "x" / (1.0 + EXP(-"x"));
    "phi" := "phi" + "w0c_14_28_1" * SIN(1 * 0.4 * "x") + "w0d_14_28_1" * COS(1 * 0.4 * "x");
    "phi" := "phi" + "w0c_14_28_2" * SIN(2 * 0.4 * "x") + "w0d_14_28_2" * COS(2 * 0.4 * "x");
    "phi" := "phi" + "w0c_14_28_3" * SIN(3 * 0.4 * "x") + "w0d_14_28_3" * COS(3 * 0.4 * "x");
    "phi" := "phi" + "w0c_14_28_4" * SIN(4 * 0.4 * "x") + "w0d_14_28_4" * COS(4 * 0.4 * "x");
    "phi" := "phi" + "w0c_14_28_5" * SIN(5 * 0.4 * "x") + "w0d_14_28_5" * COS(5 * 0.4 * "x");
    "phi" := "phi" + "w0c_14_28_6" * SIN(6 * 0.4 * "x") + "w0d_14_28_6" * COS(6 * 0.4 * "x");
    "acc" := "acc" + "phi";
    "h1_14" := "acc" + "b0_14";
    "acc" := 0.0;
    "x" := "feat_1";
    "phi" := "w0b_15_1" * "x" / (1.0 + EXP(-"x"));
    "phi" := "phi" + "w0c_15_1_1" * SIN(1 * 0.4 * "x") + "w0d_15_1_1" * COS(1 * 0.4 * "x");
    "phi" := "phi" + "w0c_15_1_2" * SIN(2 * 0.4 * "x") + "w0d_15_1_2" * COS(2 * 0.4 * "x");
    "phi" := "phi" + "w0c_15_1_3" * SIN(3 * 0.4 * "x") + "w0d_15_1_3" * COS(3 * 0.4 * "x");
    "phi" := "phi" + "w0c_15_1_4" * SIN(4 * 0.4 * "x") + "w0d_15_1_4" * COS(4 * 0.4 * "x");
    "phi" := "phi" + "w0c_15_1_5" * SIN(5 * 0.4 * "x") + "w0d_15_1_5" * COS(5 * 0.4 * "x");
    "phi" := "phi" + "w0c_15_1_6" * SIN(6 * 0.4 * "x") + "w0d_15_1_6" * COS(6 * 0.4 * "x");
    "acc" := "acc" + "phi";
    "x" := "feat_2";
    "phi" := "w0b_15_2" * "x" / (1.0 + EXP(-"x"));
    "phi" := "phi" + "w0c_15_2_1" * SIN(1 * 0.4 * "x") + "w0d_15_2_1" * COS(1 * 0.4 * "x");
    "phi" := "phi" + "w0c_15_2_2" * SIN(2 * 0.4 * "x") + "w0d_15_2_2" * COS(2 * 0.4 * "x");
    "phi" := "phi" + "w0c_15_2_3" * SIN(3 * 0.4 * "x") + "w0d_15_2_3" * COS(3 * 0.4 * "x");
    "phi" := "phi" + "w0c_15_2_4" * SIN(4 * 0.4 * "x") + "w0d_15_2_4" * COS(4 * 0.4 * "x");
    "phi" := "phi" + "w0c_15_2_5" * SIN(5 * 0.4 * "x") + "w0d_15_2_5" * COS(5 * 0.4 * "x");
    "phi" := "phi" + "w0c_15_2_6" * SIN(6 * 0.4 * "x") + "w0d_15_2_6" * COS(6 * 0.4 * "x");
    "acc" := "acc" + "phi";
    "x" := "feat_3";
    "phi" := "w0b_15_3" * "x" / (1.0 + EXP(-"x"));
    "phi" := "phi" + "w0c_15_3_1" * SIN(1 * 0.4 * "x") + "w0d_15_3_1" * COS(1 * 0.4 * "x");
    "phi" := "phi" + "w0c_15_3_2" * SIN(2 * 0.4 * "x") + "w0d_15_3_2" * COS(2 * 0.4 * "x");
    "phi" := "phi" + "w0c_15_3_3" * SIN(3 * 0.4 * "x") + "w0d_15_3_3" * COS(3 * 0.4 * "x");
    "phi" := "phi" + "w0c_15_3_4" * SIN(4 * 0.4 * "x") + "w0d_15_3_4" * COS(4 * 0.4 * "x");
    "phi" := "phi" + "w0c_15_3_5" * SIN(5 * 0.4 * "x") + "w0d_15_3_5" * COS(5 * 0.4 * "x");
    "phi" := "phi" + "w0c_15_3_6" * SIN(6 * 0.4 * "x") + "w0d_15_3_6" * COS(6 * 0.4 * "x");
    "acc" := "acc" + "phi";
    "x" := "feat_4";
    "phi" := "w0b_15_4" * "x" / (1.0 + EXP(-"x"));
    "phi" := "phi" + "w0c_15_4_1" * SIN(1 * 0.4 * "x") + "w0d_15_4_1" * COS(1 * 0.4 * "x");
    "phi" := "phi" + "w0c_15_4_2" * SIN(2 * 0.4 * "x") + "w0d_15_4_2" * COS(2 * 0.4 * "x");
    "phi" := "phi" + "w0c_15_4_3" * SIN(3 * 0.4 * "x") + "w0d_15_4_3" * COS(3 * 0.4 * "x");
    "phi" := "phi" + "w0c_15_4_4" * SIN(4 * 0.4 * "x") + "w0d_15_4_4" * COS(4 * 0.4 * "x");
    "phi" := "phi" + "w0c_15_4_5" * SIN(5 * 0.4 * "x") + "w0d_15_4_5" * COS(5 * 0.4 * "x");
    "phi" := "phi" + "w0c_15_4_6" * SIN(6 * 0.4 * "x") + "w0d_15_4_6" * COS(6 * 0.4 * "x");
    "acc" := "acc" + "phi";
    "x" := "feat_5";
    "phi" := "w0b_15_5" * "x" / (1.0 + EXP(-"x"));
    "phi" := "phi" + "w0c_15_5_1" * SIN(1 * 0.4 * "x") + "w0d_15_5_1" * COS(1 * 0.4 * "x");
    "phi" := "phi" + "w0c_15_5_2" * SIN(2 * 0.4 * "x") + "w0d_15_5_2" * COS(2 * 0.4 * "x");
    "phi" := "phi" + "w0c_15_5_3" * SIN(3 * 0.4 * "x") + "w0d_15_5_3" * COS(3 * 0.4 * "x");
    "phi" := "phi" + "w0c_15_5_4" * SIN(4 * 0.4 * "x") + "w0d_15_5_4" * COS(4 * 0.4 * "x");
    "phi" := "phi" + "w0c_15_5_5" * SIN(5 * 0.4 * "x") + "w0d_15_5_5" * COS(5 * 0.4 * "x");
    "phi" := "phi" + "w0c_15_5_6" * SIN(6 * 0.4 * "x") + "w0d_15_5_6" * COS(6 * 0.4 * "x");
    "acc" := "acc" + "phi";
    "x" := "feat_6";
    "phi" := "w0b_15_6" * "x" / (1.0 + EXP(-"x"));
    "phi" := "phi" + "w0c_15_6_1" * SIN(1 * 0.4 * "x") + "w0d_15_6_1" * COS(1 * 0.4 * "x");
    "phi" := "phi" + "w0c_15_6_2" * SIN(2 * 0.4 * "x") + "w0d_15_6_2" * COS(2 * 0.4 * "x");
    "phi" := "phi" + "w0c_15_6_3" * SIN(3 * 0.4 * "x") + "w0d_15_6_3" * COS(3 * 0.4 * "x");
    "phi" := "phi" + "w0c_15_6_4" * SIN(4 * 0.4 * "x") + "w0d_15_6_4" * COS(4 * 0.4 * "x");
    "phi" := "phi" + "w0c_15_6_5" * SIN(5 * 0.4 * "x") + "w0d_15_6_5" * COS(5 * 0.4 * "x");
    "phi" := "phi" + "w0c_15_6_6" * SIN(6 * 0.4 * "x") + "w0d_15_6_6" * COS(6 * 0.4 * "x");
    "acc" := "acc" + "phi";
    "x" := "feat_7";
    "phi" := "w0b_15_7" * "x" / (1.0 + EXP(-"x"));
    "phi" := "phi" + "w0c_15_7_1" * SIN(1 * 0.4 * "x") + "w0d_15_7_1" * COS(1 * 0.4 * "x");
    "phi" := "phi" + "w0c_15_7_2" * SIN(2 * 0.4 * "x") + "w0d_15_7_2" * COS(2 * 0.4 * "x");
    "phi" := "phi" + "w0c_15_7_3" * SIN(3 * 0.4 * "x") + "w0d_15_7_3" * COS(3 * 0.4 * "x");
    "phi" := "phi" + "w0c_15_7_4" * SIN(4 * 0.4 * "x") + "w0d_15_7_4" * COS(4 * 0.4 * "x");
    "phi" := "phi" + "w0c_15_7_5" * SIN(5 * 0.4 * "x") + "w0d_15_7_5" * COS(5 * 0.4 * "x");
    "phi" := "phi" + "w0c_15_7_6" * SIN(6 * 0.4 * "x") + "w0d_15_7_6" * COS(6 * 0.4 * "x");
    "acc" := "acc" + "phi";
    "x" := "feat_8";
    "phi" := "w0b_15_8" * "x" / (1.0 + EXP(-"x"));
    "phi" := "phi" + "w0c_15_8_1" * SIN(1 * 0.4 * "x") + "w0d_15_8_1" * COS(1 * 0.4 * "x");
    "phi" := "phi" + "w0c_15_8_2" * SIN(2 * 0.4 * "x") + "w0d_15_8_2" * COS(2 * 0.4 * "x");
    "phi" := "phi" + "w0c_15_8_3" * SIN(3 * 0.4 * "x") + "w0d_15_8_3" * COS(3 * 0.4 * "x");
    "phi" := "phi" + "w0c_15_8_4" * SIN(4 * 0.4 * "x") + "w0d_15_8_4" * COS(4 * 0.4 * "x");
    "phi" := "phi" + "w0c_15_8_5" * SIN(5 * 0.4 * "x") + "w0d_15_8_5" * COS(5 * 0.4 * "x");
    "phi" := "phi" + "w0c_15_8_6" * SIN(6 * 0.4 * "x") + "w0d_15_8_6" * COS(6 * 0.4 * "x");
    "acc" := "acc" + "phi";
    "x" := "feat_9";
    "phi" := "w0b_15_9" * "x" / (1.0 + EXP(-"x"));
    "phi" := "phi" + "w0c_15_9_1" * SIN(1 * 0.4 * "x") + "w0d_15_9_1" * COS(1 * 0.4 * "x");
    "phi" := "phi" + "w0c_15_9_2" * SIN(2 * 0.4 * "x") + "w0d_15_9_2" * COS(2 * 0.4 * "x");
    "phi" := "phi" + "w0c_15_9_3" * SIN(3 * 0.4 * "x") + "w0d_15_9_3" * COS(3 * 0.4 * "x");
    "phi" := "phi" + "w0c_15_9_4" * SIN(4 * 0.4 * "x") + "w0d_15_9_4" * COS(4 * 0.4 * "x");
    "phi" := "phi" + "w0c_15_9_5" * SIN(5 * 0.4 * "x") + "w0d_15_9_5" * COS(5 * 0.4 * "x");
    "phi" := "phi" + "w0c_15_9_6" * SIN(6 * 0.4 * "x") + "w0d_15_9_6" * COS(6 * 0.4 * "x");
    "acc" := "acc" + "phi";
    "x" := "feat_10";
    "phi" := "w0b_15_10" * "x" / (1.0 + EXP(-"x"));
    "phi" := "phi" + "w0c_15_10_1" * SIN(1 * 0.4 * "x") + "w0d_15_10_1" * COS(1 * 0.4 * "x");
    "phi" := "phi" + "w0c_15_10_2" * SIN(2 * 0.4 * "x") + "w0d_15_10_2" * COS(2 * 0.4 * "x");
    "phi" := "phi" + "w0c_15_10_3" * SIN(3 * 0.4 * "x") + "w0d_15_10_3" * COS(3 * 0.4 * "x");
    "phi" := "phi" + "w0c_15_10_4" * SIN(4 * 0.4 * "x") + "w0d_15_10_4" * COS(4 * 0.4 * "x");
    "phi" := "phi" + "w0c_15_10_5" * SIN(5 * 0.4 * "x") + "w0d_15_10_5" * COS(5 * 0.4 * "x");
    "phi" := "phi" + "w0c_15_10_6" * SIN(6 * 0.4 * "x") + "w0d_15_10_6" * COS(6 * 0.4 * "x");
    "acc" := "acc" + "phi";
    "x" := "feat_11";
    "phi" := "w0b_15_11" * "x" / (1.0 + EXP(-"x"));
    "phi" := "phi" + "w0c_15_11_1" * SIN(1 * 0.4 * "x") + "w0d_15_11_1" * COS(1 * 0.4 * "x");
    "phi" := "phi" + "w0c_15_11_2" * SIN(2 * 0.4 * "x") + "w0d_15_11_2" * COS(2 * 0.4 * "x");
    "phi" := "phi" + "w0c_15_11_3" * SIN(3 * 0.4 * "x") + "w0d_15_11_3" * COS(3 * 0.4 * "x");
    "phi" := "phi" + "w0c_15_11_4" * SIN(4 * 0.4 * "x") + "w0d_15_11_4" * COS(4 * 0.4 * "x");
    "phi" := "phi" + "w0c_15_11_5" * SIN(5 * 0.4 * "x") + "w0d_15_11_5" * COS(5 * 0.4 * "x");
    "phi" := "phi" + "w0c_15_11_6" * SIN(6 * 0.4 * "x") + "w0d_15_11_6" * COS(6 * 0.4 * "x");
    "acc" := "acc" + "phi";
    "x" := "feat_12";
    "phi" := "w0b_15_12" * "x" / (1.0 + EXP(-"x"));
    "phi" := "phi" + "w0c_15_12_1" * SIN(1 * 0.4 * "x") + "w0d_15_12_1" * COS(1 * 0.4 * "x");
    "phi" := "phi" + "w0c_15_12_2" * SIN(2 * 0.4 * "x") + "w0d_15_12_2" * COS(2 * 0.4 * "x");
    "phi" := "phi" + "w0c_15_12_3" * SIN(3 * 0.4 * "x") + "w0d_15_12_3" * COS(3 * 0.4 * "x");
    "phi" := "phi" + "w0c_15_12_4" * SIN(4 * 0.4 * "x") + "w0d_15_12_4" * COS(4 * 0.4 * "x");
    "phi" := "phi" + "w0c_15_12_5" * SIN(5 * 0.4 * "x") + "w0d_15_12_5" * COS(5 * 0.4 * "x");
    "phi" := "phi" + "w0c_15_12_6" * SIN(6 * 0.4 * "x") + "w0d_15_12_6" * COS(6 * 0.4 * "x");
    "acc" := "acc" + "phi";
    "x" := "feat_13";
    "phi" := "w0b_15_13" * "x" / (1.0 + EXP(-"x"));
    "phi" := "phi" + "w0c_15_13_1" * SIN(1 * 0.4 * "x") + "w0d_15_13_1" * COS(1 * 0.4 * "x");
    "phi" := "phi" + "w0c_15_13_2" * SIN(2 * 0.4 * "x") + "w0d_15_13_2" * COS(2 * 0.4 * "x");
    "phi" := "phi" + "w0c_15_13_3" * SIN(3 * 0.4 * "x") + "w0d_15_13_3" * COS(3 * 0.4 * "x");
    "phi" := "phi" + "w0c_15_13_4" * SIN(4 * 0.4 * "x") + "w0d_15_13_4" * COS(4 * 0.4 * "x");
    "phi" := "phi" + "w0c_15_13_5" * SIN(5 * 0.4 * "x") + "w0d_15_13_5" * COS(5 * 0.4 * "x");
    "phi" := "phi" + "w0c_15_13_6" * SIN(6 * 0.4 * "x") + "w0d_15_13_6" * COS(6 * 0.4 * "x");
    "acc" := "acc" + "phi";
    "x" := "feat_14";
    "phi" := "w0b_15_14" * "x" / (1.0 + EXP(-"x"));
    "phi" := "phi" + "w0c_15_14_1" * SIN(1 * 0.4 * "x") + "w0d_15_14_1" * COS(1 * 0.4 * "x");
    "phi" := "phi" + "w0c_15_14_2" * SIN(2 * 0.4 * "x") + "w0d_15_14_2" * COS(2 * 0.4 * "x");
    "phi" := "phi" + "w0c_15_14_3" * SIN(3 * 0.4 * "x") + "w0d_15_14_3" * COS(3 * 0.4 * "x");
    "phi" := "phi" + "w0c_15_14_4" * SIN(4 * 0.4 * "x") + "w0d_15_14_4" * COS(4 * 0.4 * "x");
    "phi" := "phi" + "w0c_15_14_5" * SIN(5 * 0.4 * "x") + "w0d_15_14_5" * COS(5 * 0.4 * "x");
    "phi" := "phi" + "w0c_15_14_6" * SIN(6 * 0.4 * "x") + "w0d_15_14_6" * COS(6 * 0.4 * "x");
    "acc" := "acc" + "phi";
    "x" := "feat_15";
    "phi" := "w0b_15_15" * "x" / (1.0 + EXP(-"x"));
    "phi" := "phi" + "w0c_15_15_1" * SIN(1 * 0.4 * "x") + "w0d_15_15_1" * COS(1 * 0.4 * "x");
    "phi" := "phi" + "w0c_15_15_2" * SIN(2 * 0.4 * "x") + "w0d_15_15_2" * COS(2 * 0.4 * "x");
    "phi" := "phi" + "w0c_15_15_3" * SIN(3 * 0.4 * "x") + "w0d_15_15_3" * COS(3 * 0.4 * "x");
    "phi" := "phi" + "w0c_15_15_4" * SIN(4 * 0.4 * "x") + "w0d_15_15_4" * COS(4 * 0.4 * "x");
    "phi" := "phi" + "w0c_15_15_5" * SIN(5 * 0.4 * "x") + "w0d_15_15_5" * COS(5 * 0.4 * "x");
    "phi" := "phi" + "w0c_15_15_6" * SIN(6 * 0.4 * "x") + "w0d_15_15_6" * COS(6 * 0.4 * "x");
    "acc" := "acc" + "phi";
    "x" := "feat_16";
    "phi" := "w0b_15_16" * "x" / (1.0 + EXP(-"x"));
    "phi" := "phi" + "w0c_15_16_1" * SIN(1 * 0.4 * "x") + "w0d_15_16_1" * COS(1 * 0.4 * "x");
    "phi" := "phi" + "w0c_15_16_2" * SIN(2 * 0.4 * "x") + "w0d_15_16_2" * COS(2 * 0.4 * "x");
    "phi" := "phi" + "w0c_15_16_3" * SIN(3 * 0.4 * "x") + "w0d_15_16_3" * COS(3 * 0.4 * "x");
    "phi" := "phi" + "w0c_15_16_4" * SIN(4 * 0.4 * "x") + "w0d_15_16_4" * COS(4 * 0.4 * "x");
    "phi" := "phi" + "w0c_15_16_5" * SIN(5 * 0.4 * "x") + "w0d_15_16_5" * COS(5 * 0.4 * "x");
    "phi" := "phi" + "w0c_15_16_6" * SIN(6 * 0.4 * "x") + "w0d_15_16_6" * COS(6 * 0.4 * "x");
    "acc" := "acc" + "phi";
    "x" := "feat_17";
    "phi" := "w0b_15_17" * "x" / (1.0 + EXP(-"x"));
    "phi" := "phi" + "w0c_15_17_1" * SIN(1 * 0.4 * "x") + "w0d_15_17_1" * COS(1 * 0.4 * "x");
    "phi" := "phi" + "w0c_15_17_2" * SIN(2 * 0.4 * "x") + "w0d_15_17_2" * COS(2 * 0.4 * "x");
    "phi" := "phi" + "w0c_15_17_3" * SIN(3 * 0.4 * "x") + "w0d_15_17_3" * COS(3 * 0.4 * "x");
    "phi" := "phi" + "w0c_15_17_4" * SIN(4 * 0.4 * "x") + "w0d_15_17_4" * COS(4 * 0.4 * "x");
    "phi" := "phi" + "w0c_15_17_5" * SIN(5 * 0.4 * "x") + "w0d_15_17_5" * COS(5 * 0.4 * "x");
    "phi" := "phi" + "w0c_15_17_6" * SIN(6 * 0.4 * "x") + "w0d_15_17_6" * COS(6 * 0.4 * "x");
    "acc" := "acc" + "phi";
    "x" := "feat_18";
    "phi" := "w0b_15_18" * "x" / (1.0 + EXP(-"x"));
    "phi" := "phi" + "w0c_15_18_1" * SIN(1 * 0.4 * "x") + "w0d_15_18_1" * COS(1 * 0.4 * "x");
    "phi" := "phi" + "w0c_15_18_2" * SIN(2 * 0.4 * "x") + "w0d_15_18_2" * COS(2 * 0.4 * "x");
    "phi" := "phi" + "w0c_15_18_3" * SIN(3 * 0.4 * "x") + "w0d_15_18_3" * COS(3 * 0.4 * "x");
    "phi" := "phi" + "w0c_15_18_4" * SIN(4 * 0.4 * "x") + "w0d_15_18_4" * COS(4 * 0.4 * "x");
    "phi" := "phi" + "w0c_15_18_5" * SIN(5 * 0.4 * "x") + "w0d_15_18_5" * COS(5 * 0.4 * "x");
    "phi" := "phi" + "w0c_15_18_6" * SIN(6 * 0.4 * "x") + "w0d_15_18_6" * COS(6 * 0.4 * "x");
    "acc" := "acc" + "phi";
    "x" := "feat_19";
    "phi" := "w0b_15_19" * "x" / (1.0 + EXP(-"x"));
    "phi" := "phi" + "w0c_15_19_1" * SIN(1 * 0.4 * "x") + "w0d_15_19_1" * COS(1 * 0.4 * "x");
    "phi" := "phi" + "w0c_15_19_2" * SIN(2 * 0.4 * "x") + "w0d_15_19_2" * COS(2 * 0.4 * "x");
    "phi" := "phi" + "w0c_15_19_3" * SIN(3 * 0.4 * "x") + "w0d_15_19_3" * COS(3 * 0.4 * "x");
    "phi" := "phi" + "w0c_15_19_4" * SIN(4 * 0.4 * "x") + "w0d_15_19_4" * COS(4 * 0.4 * "x");
    "phi" := "phi" + "w0c_15_19_5" * SIN(5 * 0.4 * "x") + "w0d_15_19_5" * COS(5 * 0.4 * "x");
    "phi" := "phi" + "w0c_15_19_6" * SIN(6 * 0.4 * "x") + "w0d_15_19_6" * COS(6 * 0.4 * "x");
    "acc" := "acc" + "phi";
    "x" := "feat_20";
    "phi" := "w0b_15_20" * "x" / (1.0 + EXP(-"x"));
    "phi" := "phi" + "w0c_15_20_1" * SIN(1 * 0.4 * "x") + "w0d_15_20_1" * COS(1 * 0.4 * "x");
    "phi" := "phi" + "w0c_15_20_2" * SIN(2 * 0.4 * "x") + "w0d_15_20_2" * COS(2 * 0.4 * "x");
    "phi" := "phi" + "w0c_15_20_3" * SIN(3 * 0.4 * "x") + "w0d_15_20_3" * COS(3 * 0.4 * "x");
    "phi" := "phi" + "w0c_15_20_4" * SIN(4 * 0.4 * "x") + "w0d_15_20_4" * COS(4 * 0.4 * "x");
    "phi" := "phi" + "w0c_15_20_5" * SIN(5 * 0.4 * "x") + "w0d_15_20_5" * COS(5 * 0.4 * "x");
    "phi" := "phi" + "w0c_15_20_6" * SIN(6 * 0.4 * "x") + "w0d_15_20_6" * COS(6 * 0.4 * "x");
    "acc" := "acc" + "phi";
    "x" := "feat_21";
    "phi" := "w0b_15_21" * "x" / (1.0 + EXP(-"x"));
    "phi" := "phi" + "w0c_15_21_1" * SIN(1 * 0.4 * "x") + "w0d_15_21_1" * COS(1 * 0.4 * "x");
    "phi" := "phi" + "w0c_15_21_2" * SIN(2 * 0.4 * "x") + "w0d_15_21_2" * COS(2 * 0.4 * "x");
    "phi" := "phi" + "w0c_15_21_3" * SIN(3 * 0.4 * "x") + "w0d_15_21_3" * COS(3 * 0.4 * "x");
    "phi" := "phi" + "w0c_15_21_4" * SIN(4 * 0.4 * "x") + "w0d_15_21_4" * COS(4 * 0.4 * "x");
    "phi" := "phi" + "w0c_15_21_5" * SIN(5 * 0.4 * "x") + "w0d_15_21_5" * COS(5 * 0.4 * "x");
    "phi" := "phi" + "w0c_15_21_6" * SIN(6 * 0.4 * "x") + "w0d_15_21_6" * COS(6 * 0.4 * "x");
    "acc" := "acc" + "phi";
    "x" := "feat_22";
    "phi" := "w0b_15_22" * "x" / (1.0 + EXP(-"x"));
    "phi" := "phi" + "w0c_15_22_1" * SIN(1 * 0.4 * "x") + "w0d_15_22_1" * COS(1 * 0.4 * "x");
    "phi" := "phi" + "w0c_15_22_2" * SIN(2 * 0.4 * "x") + "w0d_15_22_2" * COS(2 * 0.4 * "x");
    "phi" := "phi" + "w0c_15_22_3" * SIN(3 * 0.4 * "x") + "w0d_15_22_3" * COS(3 * 0.4 * "x");
    "phi" := "phi" + "w0c_15_22_4" * SIN(4 * 0.4 * "x") + "w0d_15_22_4" * COS(4 * 0.4 * "x");
    "phi" := "phi" + "w0c_15_22_5" * SIN(5 * 0.4 * "x") + "w0d_15_22_5" * COS(5 * 0.4 * "x");
    "phi" := "phi" + "w0c_15_22_6" * SIN(6 * 0.4 * "x") + "w0d_15_22_6" * COS(6 * 0.4 * "x");
    "acc" := "acc" + "phi";
    "x" := "feat_23";
    "phi" := "w0b_15_23" * "x" / (1.0 + EXP(-"x"));
    "phi" := "phi" + "w0c_15_23_1" * SIN(1 * 0.4 * "x") + "w0d_15_23_1" * COS(1 * 0.4 * "x");
    "phi" := "phi" + "w0c_15_23_2" * SIN(2 * 0.4 * "x") + "w0d_15_23_2" * COS(2 * 0.4 * "x");
    "phi" := "phi" + "w0c_15_23_3" * SIN(3 * 0.4 * "x") + "w0d_15_23_3" * COS(3 * 0.4 * "x");
    "phi" := "phi" + "w0c_15_23_4" * SIN(4 * 0.4 * "x") + "w0d_15_23_4" * COS(4 * 0.4 * "x");
    "phi" := "phi" + "w0c_15_23_5" * SIN(5 * 0.4 * "x") + "w0d_15_23_5" * COS(5 * 0.4 * "x");
    "phi" := "phi" + "w0c_15_23_6" * SIN(6 * 0.4 * "x") + "w0d_15_23_6" * COS(6 * 0.4 * "x");
    "acc" := "acc" + "phi";
    "x" := "feat_24";
    "phi" := "w0b_15_24" * "x" / (1.0 + EXP(-"x"));
    "phi" := "phi" + "w0c_15_24_1" * SIN(1 * 0.4 * "x") + "w0d_15_24_1" * COS(1 * 0.4 * "x");
    "phi" := "phi" + "w0c_15_24_2" * SIN(2 * 0.4 * "x") + "w0d_15_24_2" * COS(2 * 0.4 * "x");
    "phi" := "phi" + "w0c_15_24_3" * SIN(3 * 0.4 * "x") + "w0d_15_24_3" * COS(3 * 0.4 * "x");
    "phi" := "phi" + "w0c_15_24_4" * SIN(4 * 0.4 * "x") + "w0d_15_24_4" * COS(4 * 0.4 * "x");
    "phi" := "phi" + "w0c_15_24_5" * SIN(5 * 0.4 * "x") + "w0d_15_24_5" * COS(5 * 0.4 * "x");
    "phi" := "phi" + "w0c_15_24_6" * SIN(6 * 0.4 * "x") + "w0d_15_24_6" * COS(6 * 0.4 * "x");
    "acc" := "acc" + "phi";
    "x" := "feat_25";
    "phi" := "w0b_15_25" * "x" / (1.0 + EXP(-"x"));
    "phi" := "phi" + "w0c_15_25_1" * SIN(1 * 0.4 * "x") + "w0d_15_25_1" * COS(1 * 0.4 * "x");
    "phi" := "phi" + "w0c_15_25_2" * SIN(2 * 0.4 * "x") + "w0d_15_25_2" * COS(2 * 0.4 * "x");
    "phi" := "phi" + "w0c_15_25_3" * SIN(3 * 0.4 * "x") + "w0d_15_25_3" * COS(3 * 0.4 * "x");
    "phi" := "phi" + "w0c_15_25_4" * SIN(4 * 0.4 * "x") + "w0d_15_25_4" * COS(4 * 0.4 * "x");
    "phi" := "phi" + "w0c_15_25_5" * SIN(5 * 0.4 * "x") + "w0d_15_25_5" * COS(5 * 0.4 * "x");
    "phi" := "phi" + "w0c_15_25_6" * SIN(6 * 0.4 * "x") + "w0d_15_25_6" * COS(6 * 0.4 * "x");
    "acc" := "acc" + "phi";
    "x" := "feat_26";
    "phi" := "w0b_15_26" * "x" / (1.0 + EXP(-"x"));
    "phi" := "phi" + "w0c_15_26_1" * SIN(1 * 0.4 * "x") + "w0d_15_26_1" * COS(1 * 0.4 * "x");
    "phi" := "phi" + "w0c_15_26_2" * SIN(2 * 0.4 * "x") + "w0d_15_26_2" * COS(2 * 0.4 * "x");
    "phi" := "phi" + "w0c_15_26_3" * SIN(3 * 0.4 * "x") + "w0d_15_26_3" * COS(3 * 0.4 * "x");
    "phi" := "phi" + "w0c_15_26_4" * SIN(4 * 0.4 * "x") + "w0d_15_26_4" * COS(4 * 0.4 * "x");
    "phi" := "phi" + "w0c_15_26_5" * SIN(5 * 0.4 * "x") + "w0d_15_26_5" * COS(5 * 0.4 * "x");
    "phi" := "phi" + "w0c_15_26_6" * SIN(6 * 0.4 * "x") + "w0d_15_26_6" * COS(6 * 0.4 * "x");
    "acc" := "acc" + "phi";
    "x" := "feat_27";
    "phi" := "w0b_15_27" * "x" / (1.0 + EXP(-"x"));
    "phi" := "phi" + "w0c_15_27_1" * SIN(1 * 0.4 * "x") + "w0d_15_27_1" * COS(1 * 0.4 * "x");
    "phi" := "phi" + "w0c_15_27_2" * SIN(2 * 0.4 * "x") + "w0d_15_27_2" * COS(2 * 0.4 * "x");
    "phi" := "phi" + "w0c_15_27_3" * SIN(3 * 0.4 * "x") + "w0d_15_27_3" * COS(3 * 0.4 * "x");
    "phi" := "phi" + "w0c_15_27_4" * SIN(4 * 0.4 * "x") + "w0d_15_27_4" * COS(4 * 0.4 * "x");
    "phi" := "phi" + "w0c_15_27_5" * SIN(5 * 0.4 * "x") + "w0d_15_27_5" * COS(5 * 0.4 * "x");
    "phi" := "phi" + "w0c_15_27_6" * SIN(6 * 0.4 * "x") + "w0d_15_27_6" * COS(6 * 0.4 * "x");
    "acc" := "acc" + "phi";
    "x" := "feat_28";
    "phi" := "w0b_15_28" * "x" / (1.0 + EXP(-"x"));
    "phi" := "phi" + "w0c_15_28_1" * SIN(1 * 0.4 * "x") + "w0d_15_28_1" * COS(1 * 0.4 * "x");
    "phi" := "phi" + "w0c_15_28_2" * SIN(2 * 0.4 * "x") + "w0d_15_28_2" * COS(2 * 0.4 * "x");
    "phi" := "phi" + "w0c_15_28_3" * SIN(3 * 0.4 * "x") + "w0d_15_28_3" * COS(3 * 0.4 * "x");
    "phi" := "phi" + "w0c_15_28_4" * SIN(4 * 0.4 * "x") + "w0d_15_28_4" * COS(4 * 0.4 * "x");
    "phi" := "phi" + "w0c_15_28_5" * SIN(5 * 0.4 * "x") + "w0d_15_28_5" * COS(5 * 0.4 * "x");
    "phi" := "phi" + "w0c_15_28_6" * SIN(6 * 0.4 * "x") + "w0d_15_28_6" * COS(6 * 0.4 * "x");
    "acc" := "acc" + "phi";
    "h1_15" := "acc" + "b0_15";
    "acc" := 0.0;
    "x" := "feat_1";
    "phi" := "w0b_16_1" * "x" / (1.0 + EXP(-"x"));
    "phi" := "phi" + "w0c_16_1_1" * SIN(1 * 0.4 * "x") + "w0d_16_1_1" * COS(1 * 0.4 * "x");
    "phi" := "phi" + "w0c_16_1_2" * SIN(2 * 0.4 * "x") + "w0d_16_1_2" * COS(2 * 0.4 * "x");
    "phi" := "phi" + "w0c_16_1_3" * SIN(3 * 0.4 * "x") + "w0d_16_1_3" * COS(3 * 0.4 * "x");
    "phi" := "phi" + "w0c_16_1_4" * SIN(4 * 0.4 * "x") + "w0d_16_1_4" * COS(4 * 0.4 * "x");
    "phi" := "phi" + "w0c_16_1_5" * SIN(5 * 0.4 * "x") + "w0d_16_1_5" * COS(5 * 0.4 * "x");
    "phi" := "phi" + "w0c_16_1_6" * SIN(6 * 0.4 * "x") + "w0d_16_1_6" * COS(6 * 0.4 * "x");
    "acc" := "acc" + "phi";
    "x" := "feat_2";
    "phi" := "w0b_16_2" * "x" / (1.0 + EXP(-"x"));
    "phi" := "phi" + "w0c_16_2_1" * SIN(1 * 0.4 * "x") + "w0d_16_2_1" * COS(1 * 0.4 * "x");
    "phi" := "phi" + "w0c_16_2_2" * SIN(2 * 0.4 * "x") + "w0d_16_2_2" * COS(2 * 0.4 * "x");
    "phi" := "phi" + "w0c_16_2_3" * SIN(3 * 0.4 * "x") + "w0d_16_2_3" * COS(3 * 0.4 * "x");
    "phi" := "phi" + "w0c_16_2_4" * SIN(4 * 0.4 * "x") + "w0d_16_2_4" * COS(4 * 0.4 * "x");
    "phi" := "phi" + "w0c_16_2_5" * SIN(5 * 0.4 * "x") + "w0d_16_2_5" * COS(5 * 0.4 * "x");
    "phi" := "phi" + "w0c_16_2_6" * SIN(6 * 0.4 * "x") + "w0d_16_2_6" * COS(6 * 0.4 * "x");
    "acc" := "acc" + "phi";
    "x" := "feat_3";
    "phi" := "w0b_16_3" * "x" / (1.0 + EXP(-"x"));
    "phi" := "phi" + "w0c_16_3_1" * SIN(1 * 0.4 * "x") + "w0d_16_3_1" * COS(1 * 0.4 * "x");
    "phi" := "phi" + "w0c_16_3_2" * SIN(2 * 0.4 * "x") + "w0d_16_3_2" * COS(2 * 0.4 * "x");
    "phi" := "phi" + "w0c_16_3_3" * SIN(3 * 0.4 * "x") + "w0d_16_3_3" * COS(3 * 0.4 * "x");
    "phi" := "phi" + "w0c_16_3_4" * SIN(4 * 0.4 * "x") + "w0d_16_3_4" * COS(4 * 0.4 * "x");
    "phi" := "phi" + "w0c_16_3_5" * SIN(5 * 0.4 * "x") + "w0d_16_3_5" * COS(5 * 0.4 * "x");
    "phi" := "phi" + "w0c_16_3_6" * SIN(6 * 0.4 * "x") + "w0d_16_3_6" * COS(6 * 0.4 * "x");
    "acc" := "acc" + "phi";
    "x" := "feat_4";
    "phi" := "w0b_16_4" * "x" / (1.0 + EXP(-"x"));
    "phi" := "phi" + "w0c_16_4_1" * SIN(1 * 0.4 * "x") + "w0d_16_4_1" * COS(1 * 0.4 * "x");
    "phi" := "phi" + "w0c_16_4_2" * SIN(2 * 0.4 * "x") + "w0d_16_4_2" * COS(2 * 0.4 * "x");
    "phi" := "phi" + "w0c_16_4_3" * SIN(3 * 0.4 * "x") + "w0d_16_4_3" * COS(3 * 0.4 * "x");
    "phi" := "phi" + "w0c_16_4_4" * SIN(4 * 0.4 * "x") + "w0d_16_4_4" * COS(4 * 0.4 * "x");
    "phi" := "phi" + "w0c_16_4_5" * SIN(5 * 0.4 * "x") + "w0d_16_4_5" * COS(5 * 0.4 * "x");
    "phi" := "phi" + "w0c_16_4_6" * SIN(6 * 0.4 * "x") + "w0d_16_4_6" * COS(6 * 0.4 * "x");
    "acc" := "acc" + "phi";
    "x" := "feat_5";
    "phi" := "w0b_16_5" * "x" / (1.0 + EXP(-"x"));
    "phi" := "phi" + "w0c_16_5_1" * SIN(1 * 0.4 * "x") + "w0d_16_5_1" * COS(1 * 0.4 * "x");
    "phi" := "phi" + "w0c_16_5_2" * SIN(2 * 0.4 * "x") + "w0d_16_5_2" * COS(2 * 0.4 * "x");
    "phi" := "phi" + "w0c_16_5_3" * SIN(3 * 0.4 * "x") + "w0d_16_5_3" * COS(3 * 0.4 * "x");
    "phi" := "phi" + "w0c_16_5_4" * SIN(4 * 0.4 * "x") + "w0d_16_5_4" * COS(4 * 0.4 * "x");
    "phi" := "phi" + "w0c_16_5_5" * SIN(5 * 0.4 * "x") + "w0d_16_5_5" * COS(5 * 0.4 * "x");
    "phi" := "phi" + "w0c_16_5_6" * SIN(6 * 0.4 * "x") + "w0d_16_5_6" * COS(6 * 0.4 * "x");
    "acc" := "acc" + "phi";
    "x" := "feat_6";
    "phi" := "w0b_16_6" * "x" / (1.0 + EXP(-"x"));
    "phi" := "phi" + "w0c_16_6_1" * SIN(1 * 0.4 * "x") + "w0d_16_6_1" * COS(1 * 0.4 * "x");
    "phi" := "phi" + "w0c_16_6_2" * SIN(2 * 0.4 * "x") + "w0d_16_6_2" * COS(2 * 0.4 * "x");
    "phi" := "phi" + "w0c_16_6_3" * SIN(3 * 0.4 * "x") + "w0d_16_6_3" * COS(3 * 0.4 * "x");
    "phi" := "phi" + "w0c_16_6_4" * SIN(4 * 0.4 * "x") + "w0d_16_6_4" * COS(4 * 0.4 * "x");
    "phi" := "phi" + "w0c_16_6_5" * SIN(5 * 0.4 * "x") + "w0d_16_6_5" * COS(5 * 0.4 * "x");
    "phi" := "phi" + "w0c_16_6_6" * SIN(6 * 0.4 * "x") + "w0d_16_6_6" * COS(6 * 0.4 * "x");
    "acc" := "acc" + "phi";
    "x" := "feat_7";
    "phi" := "w0b_16_7" * "x" / (1.0 + EXP(-"x"));
    "phi" := "phi" + "w0c_16_7_1" * SIN(1 * 0.4 * "x") + "w0d_16_7_1" * COS(1 * 0.4 * "x");
    "phi" := "phi" + "w0c_16_7_2" * SIN(2 * 0.4 * "x") + "w0d_16_7_2" * COS(2 * 0.4 * "x");
    "phi" := "phi" + "w0c_16_7_3" * SIN(3 * 0.4 * "x") + "w0d_16_7_3" * COS(3 * 0.4 * "x");
    "phi" := "phi" + "w0c_16_7_4" * SIN(4 * 0.4 * "x") + "w0d_16_7_4" * COS(4 * 0.4 * "x");
    "phi" := "phi" + "w0c_16_7_5" * SIN(5 * 0.4 * "x") + "w0d_16_7_5" * COS(5 * 0.4 * "x");
    "phi" := "phi" + "w0c_16_7_6" * SIN(6 * 0.4 * "x") + "w0d_16_7_6" * COS(6 * 0.4 * "x");
    "acc" := "acc" + "phi";
    "x" := "feat_8";
    "phi" := "w0b_16_8" * "x" / (1.0 + EXP(-"x"));
    "phi" := "phi" + "w0c_16_8_1" * SIN(1 * 0.4 * "x") + "w0d_16_8_1" * COS(1 * 0.4 * "x");
    "phi" := "phi" + "w0c_16_8_2" * SIN(2 * 0.4 * "x") + "w0d_16_8_2" * COS(2 * 0.4 * "x");
    "phi" := "phi" + "w0c_16_8_3" * SIN(3 * 0.4 * "x") + "w0d_16_8_3" * COS(3 * 0.4 * "x");
    "phi" := "phi" + "w0c_16_8_4" * SIN(4 * 0.4 * "x") + "w0d_16_8_4" * COS(4 * 0.4 * "x");
    "phi" := "phi" + "w0c_16_8_5" * SIN(5 * 0.4 * "x") + "w0d_16_8_5" * COS(5 * 0.4 * "x");
    "phi" := "phi" + "w0c_16_8_6" * SIN(6 * 0.4 * "x") + "w0d_16_8_6" * COS(6 * 0.4 * "x");
    "acc" := "acc" + "phi";
    "x" := "feat_9";
    "phi" := "w0b_16_9" * "x" / (1.0 + EXP(-"x"));
    "phi" := "phi" + "w0c_16_9_1" * SIN(1 * 0.4 * "x") + "w0d_16_9_1" * COS(1 * 0.4 * "x");
    "phi" := "phi" + "w0c_16_9_2" * SIN(2 * 0.4 * "x") + "w0d_16_9_2" * COS(2 * 0.4 * "x");
    "phi" := "phi" + "w0c_16_9_3" * SIN(3 * 0.4 * "x") + "w0d_16_9_3" * COS(3 * 0.4 * "x");
    "phi" := "phi" + "w0c_16_9_4" * SIN(4 * 0.4 * "x") + "w0d_16_9_4" * COS(4 * 0.4 * "x");
    "phi" := "phi" + "w0c_16_9_5" * SIN(5 * 0.4 * "x") + "w0d_16_9_5" * COS(5 * 0.4 * "x");
    "phi" := "phi" + "w0c_16_9_6" * SIN(6 * 0.4 * "x") + "w0d_16_9_6" * COS(6 * 0.4 * "x");
    "acc" := "acc" + "phi";
    "x" := "feat_10";
    "phi" := "w0b_16_10" * "x" / (1.0 + EXP(-"x"));
    "phi" := "phi" + "w0c_16_10_1" * SIN(1 * 0.4 * "x") + "w0d_16_10_1" * COS(1 * 0.4 * "x");
    "phi" := "phi" + "w0c_16_10_2" * SIN(2 * 0.4 * "x") + "w0d_16_10_2" * COS(2 * 0.4 * "x");
    "phi" := "phi" + "w0c_16_10_3" * SIN(3 * 0.4 * "x") + "w0d_16_10_3" * COS(3 * 0.4 * "x");
    "phi" := "phi" + "w0c_16_10_4" * SIN(4 * 0.4 * "x") + "w0d_16_10_4" * COS(4 * 0.4 * "x");
    "phi" := "phi" + "w0c_16_10_5" * SIN(5 * 0.4 * "x") + "w0d_16_10_5" * COS(5 * 0.4 * "x");
    "phi" := "phi" + "w0c_16_10_6" * SIN(6 * 0.4 * "x") + "w0d_16_10_6" * COS(6 * 0.4 * "x");
    "acc" := "acc" + "phi";
    "x" := "feat_11";
    "phi" := "w0b_16_11" * "x" / (1.0 + EXP(-"x"));
    "phi" := "phi" + "w0c_16_11_1" * SIN(1 * 0.4 * "x") + "w0d_16_11_1" * COS(1 * 0.4 * "x");
    "phi" := "phi" + "w0c_16_11_2" * SIN(2 * 0.4 * "x") + "w0d_16_11_2" * COS(2 * 0.4 * "x");
    "phi" := "phi" + "w0c_16_11_3" * SIN(3 * 0.4 * "x") + "w0d_16_11_3" * COS(3 * 0.4 * "x");
    "phi" := "phi" + "w0c_16_11_4" * SIN(4 * 0.4 * "x") + "w0d_16_11_4" * COS(4 * 0.4 * "x");
    "phi" := "phi" + "w0c_16_11_5" * SIN(5 * 0.4 * "x") + "w0d_16_11_5" * COS(5 * 0.4 * "x");
    "phi" := "phi" + "w0c_16_11_6" * SIN(6 * 0.4 * "x") + "w0d_16_11_6" * COS(6 * 0.4 * "x");
    "acc" := "acc" + "phi";
    "x" := "feat_12";
    "phi" := "w0b_16_12" * "x" / (1.0 + EXP(-"x"));
    "phi" := "phi" + "w0c_16_12_1" * SIN(1 * 0.4 * "x") + "w0d_16_12_1" * COS(1 * 0.4 * "x");
    "phi" := "phi" + "w0c_16_12_2" * SIN(2 * 0.4 * "x") + "w0d_16_12_2" * COS(2 * 0.4 * "x");
    "phi" := "phi" + "w0c_16_12_3" * SIN(3 * 0.4 * "x") + "w0d_16_12_3" * COS(3 * 0.4 * "x");
    "phi" := "phi" + "w0c_16_12_4" * SIN(4 * 0.4 * "x") + "w0d_16_12_4" * COS(4 * 0.4 * "x");
    "phi" := "phi" + "w0c_16_12_5" * SIN(5 * 0.4 * "x") + "w0d_16_12_5" * COS(5 * 0.4 * "x");
    "phi" := "phi" + "w0c_16_12_6" * SIN(6 * 0.4 * "x") + "w0d_16_12_6" * COS(6 * 0.4 * "x");
    "acc" := "acc" + "phi";
    "x" := "feat_13";
    "phi" := "w0b_16_13" * "x" / (1.0 + EXP(-"x"));
    "phi" := "phi" + "w0c_16_13_1" * SIN(1 * 0.4 * "x") + "w0d_16_13_1" * COS(1 * 0.4 * "x");
    "phi" := "phi" + "w0c_16_13_2" * SIN(2 * 0.4 * "x") + "w0d_16_13_2" * COS(2 * 0.4 * "x");
    "phi" := "phi" + "w0c_16_13_3" * SIN(3 * 0.4 * "x") + "w0d_16_13_3" * COS(3 * 0.4 * "x");
    "phi" := "phi" + "w0c_16_13_4" * SIN(4 * 0.4 * "x") + "w0d_16_13_4" * COS(4 * 0.4 * "x");
    "phi" := "phi" + "w0c_16_13_5" * SIN(5 * 0.4 * "x") + "w0d_16_13_5" * COS(5 * 0.4 * "x");
    "phi" := "phi" + "w0c_16_13_6" * SIN(6 * 0.4 * "x") + "w0d_16_13_6" * COS(6 * 0.4 * "x");
    "acc" := "acc" + "phi";
    "x" := "feat_14";
    "phi" := "w0b_16_14" * "x" / (1.0 + EXP(-"x"));
    "phi" := "phi" + "w0c_16_14_1" * SIN(1 * 0.4 * "x") + "w0d_16_14_1" * COS(1 * 0.4 * "x");
    "phi" := "phi" + "w0c_16_14_2" * SIN(2 * 0.4 * "x") + "w0d_16_14_2" * COS(2 * 0.4 * "x");
    "phi" := "phi" + "w0c_16_14_3" * SIN(3 * 0.4 * "x") + "w0d_16_14_3" * COS(3 * 0.4 * "x");
    "phi" := "phi" + "w0c_16_14_4" * SIN(4 * 0.4 * "x") + "w0d_16_14_4" * COS(4 * 0.4 * "x");
    "phi" := "phi" + "w0c_16_14_5" * SIN(5 * 0.4 * "x") + "w0d_16_14_5" * COS(5 * 0.4 * "x");
    "phi" := "phi" + "w0c_16_14_6" * SIN(6 * 0.4 * "x") + "w0d_16_14_6" * COS(6 * 0.4 * "x");
    "acc" := "acc" + "phi";
    "x" := "feat_15";
    "phi" := "w0b_16_15" * "x" / (1.0 + EXP(-"x"));
    "phi" := "phi" + "w0c_16_15_1" * SIN(1 * 0.4 * "x") + "w0d_16_15_1" * COS(1 * 0.4 * "x");
    "phi" := "phi" + "w0c_16_15_2" * SIN(2 * 0.4 * "x") + "w0d_16_15_2" * COS(2 * 0.4 * "x");
    "phi" := "phi" + "w0c_16_15_3" * SIN(3 * 0.4 * "x") + "w0d_16_15_3" * COS(3 * 0.4 * "x");
    "phi" := "phi" + "w0c_16_15_4" * SIN(4 * 0.4 * "x") + "w0d_16_15_4" * COS(4 * 0.4 * "x");
    "phi" := "phi" + "w0c_16_15_5" * SIN(5 * 0.4 * "x") + "w0d_16_15_5" * COS(5 * 0.4 * "x");
    "phi" := "phi" + "w0c_16_15_6" * SIN(6 * 0.4 * "x") + "w0d_16_15_6" * COS(6 * 0.4 * "x");
    "acc" := "acc" + "phi";
    "x" := "feat_16";
    "phi" := "w0b_16_16" * "x" / (1.0 + EXP(-"x"));
    "phi" := "phi" + "w0c_16_16_1" * SIN(1 * 0.4 * "x") + "w0d_16_16_1" * COS(1 * 0.4 * "x");
    "phi" := "phi" + "w0c_16_16_2" * SIN(2 * 0.4 * "x") + "w0d_16_16_2" * COS(2 * 0.4 * "x");
    "phi" := "phi" + "w0c_16_16_3" * SIN(3 * 0.4 * "x") + "w0d_16_16_3" * COS(3 * 0.4 * "x");
    "phi" := "phi" + "w0c_16_16_4" * SIN(4 * 0.4 * "x") + "w0d_16_16_4" * COS(4 * 0.4 * "x");
    "phi" := "phi" + "w0c_16_16_5" * SIN(5 * 0.4 * "x") + "w0d_16_16_5" * COS(5 * 0.4 * "x");
    "phi" := "phi" + "w0c_16_16_6" * SIN(6 * 0.4 * "x") + "w0d_16_16_6" * COS(6 * 0.4 * "x");
    "acc" := "acc" + "phi";
    "x" := "feat_17";
    "phi" := "w0b_16_17" * "x" / (1.0 + EXP(-"x"));
    "phi" := "phi" + "w0c_16_17_1" * SIN(1 * 0.4 * "x") + "w0d_16_17_1" * COS(1 * 0.4 * "x");
    "phi" := "phi" + "w0c_16_17_2" * SIN(2 * 0.4 * "x") + "w0d_16_17_2" * COS(2 * 0.4 * "x");
    "phi" := "phi" + "w0c_16_17_3" * SIN(3 * 0.4 * "x") + "w0d_16_17_3" * COS(3 * 0.4 * "x");
    "phi" := "phi" + "w0c_16_17_4" * SIN(4 * 0.4 * "x") + "w0d_16_17_4" * COS(4 * 0.4 * "x");
    "phi" := "phi" + "w0c_16_17_5" * SIN(5 * 0.4 * "x") + "w0d_16_17_5" * COS(5 * 0.4 * "x");
    "phi" := "phi" + "w0c_16_17_6" * SIN(6 * 0.4 * "x") + "w0d_16_17_6" * COS(6 * 0.4 * "x");
    "acc" := "acc" + "phi";
    "x" := "feat_18";
    "phi" := "w0b_16_18" * "x" / (1.0 + EXP(-"x"));
    "phi" := "phi" + "w0c_16_18_1" * SIN(1 * 0.4 * "x") + "w0d_16_18_1" * COS(1 * 0.4 * "x");
    "phi" := "phi" + "w0c_16_18_2" * SIN(2 * 0.4 * "x") + "w0d_16_18_2" * COS(2 * 0.4 * "x");
    "phi" := "phi" + "w0c_16_18_3" * SIN(3 * 0.4 * "x") + "w0d_16_18_3" * COS(3 * 0.4 * "x");
    "phi" := "phi" + "w0c_16_18_4" * SIN(4 * 0.4 * "x") + "w0d_16_18_4" * COS(4 * 0.4 * "x");
    "phi" := "phi" + "w0c_16_18_5" * SIN(5 * 0.4 * "x") + "w0d_16_18_5" * COS(5 * 0.4 * "x");
    "phi" := "phi" + "w0c_16_18_6" * SIN(6 * 0.4 * "x") + "w0d_16_18_6" * COS(6 * 0.4 * "x");
    "acc" := "acc" + "phi";
    "x" := "feat_19";
    "phi" := "w0b_16_19" * "x" / (1.0 + EXP(-"x"));
    "phi" := "phi" + "w0c_16_19_1" * SIN(1 * 0.4 * "x") + "w0d_16_19_1" * COS(1 * 0.4 * "x");
    "phi" := "phi" + "w0c_16_19_2" * SIN(2 * 0.4 * "x") + "w0d_16_19_2" * COS(2 * 0.4 * "x");
    "phi" := "phi" + "w0c_16_19_3" * SIN(3 * 0.4 * "x") + "w0d_16_19_3" * COS(3 * 0.4 * "x");
    "phi" := "phi" + "w0c_16_19_4" * SIN(4 * 0.4 * "x") + "w0d_16_19_4" * COS(4 * 0.4 * "x");
    "phi" := "phi" + "w0c_16_19_5" * SIN(5 * 0.4 * "x") + "w0d_16_19_5" * COS(5 * 0.4 * "x");
    "phi" := "phi" + "w0c_16_19_6" * SIN(6 * 0.4 * "x") + "w0d_16_19_6" * COS(6 * 0.4 * "x");
    "acc" := "acc" + "phi";
    "x" := "feat_20";
    "phi" := "w0b_16_20" * "x" / (1.0 + EXP(-"x"));
    "phi" := "phi" + "w0c_16_20_1" * SIN(1 * 0.4 * "x") + "w0d_16_20_1" * COS(1 * 0.4 * "x");
    "phi" := "phi" + "w0c_16_20_2" * SIN(2 * 0.4 * "x") + "w0d_16_20_2" * COS(2 * 0.4 * "x");
    "phi" := "phi" + "w0c_16_20_3" * SIN(3 * 0.4 * "x") + "w0d_16_20_3" * COS(3 * 0.4 * "x");
    "phi" := "phi" + "w0c_16_20_4" * SIN(4 * 0.4 * "x") + "w0d_16_20_4" * COS(4 * 0.4 * "x");
    "phi" := "phi" + "w0c_16_20_5" * SIN(5 * 0.4 * "x") + "w0d_16_20_5" * COS(5 * 0.4 * "x");
    "phi" := "phi" + "w0c_16_20_6" * SIN(6 * 0.4 * "x") + "w0d_16_20_6" * COS(6 * 0.4 * "x");
    "acc" := "acc" + "phi";
    "x" := "feat_21";
    "phi" := "w0b_16_21" * "x" / (1.0 + EXP(-"x"));
    "phi" := "phi" + "w0c_16_21_1" * SIN(1 * 0.4 * "x") + "w0d_16_21_1" * COS(1 * 0.4 * "x");
    "phi" := "phi" + "w0c_16_21_2" * SIN(2 * 0.4 * "x") + "w0d_16_21_2" * COS(2 * 0.4 * "x");
    "phi" := "phi" + "w0c_16_21_3" * SIN(3 * 0.4 * "x") + "w0d_16_21_3" * COS(3 * 0.4 * "x");
    "phi" := "phi" + "w0c_16_21_4" * SIN(4 * 0.4 * "x") + "w0d_16_21_4" * COS(4 * 0.4 * "x");
    "phi" := "phi" + "w0c_16_21_5" * SIN(5 * 0.4 * "x") + "w0d_16_21_5" * COS(5 * 0.4 * "x");
    "phi" := "phi" + "w0c_16_21_6" * SIN(6 * 0.4 * "x") + "w0d_16_21_6" * COS(6 * 0.4 * "x");
    "acc" := "acc" + "phi";
    "x" := "feat_22";
    "phi" := "w0b_16_22" * "x" / (1.0 + EXP(-"x"));
    "phi" := "phi" + "w0c_16_22_1" * SIN(1 * 0.4 * "x") + "w0d_16_22_1" * COS(1 * 0.4 * "x");
    "phi" := "phi" + "w0c_16_22_2" * SIN(2 * 0.4 * "x") + "w0d_16_22_2" * COS(2 * 0.4 * "x");
    "phi" := "phi" + "w0c_16_22_3" * SIN(3 * 0.4 * "x") + "w0d_16_22_3" * COS(3 * 0.4 * "x");
    "phi" := "phi" + "w0c_16_22_4" * SIN(4 * 0.4 * "x") + "w0d_16_22_4" * COS(4 * 0.4 * "x");
    "phi" := "phi" + "w0c_16_22_5" * SIN(5 * 0.4 * "x") + "w0d_16_22_5" * COS(5 * 0.4 * "x");
    "phi" := "phi" + "w0c_16_22_6" * SIN(6 * 0.4 * "x") + "w0d_16_22_6" * COS(6 * 0.4 * "x");
    "acc" := "acc" + "phi";
    "x" := "feat_23";
    "phi" := "w0b_16_23" * "x" / (1.0 + EXP(-"x"));
    "phi" := "phi" + "w0c_16_23_1" * SIN(1 * 0.4 * "x") + "w0d_16_23_1" * COS(1 * 0.4 * "x");
    "phi" := "phi" + "w0c_16_23_2" * SIN(2 * 0.4 * "x") + "w0d_16_23_2" * COS(2 * 0.4 * "x");
    "phi" := "phi" + "w0c_16_23_3" * SIN(3 * 0.4 * "x") + "w0d_16_23_3" * COS(3 * 0.4 * "x");
    "phi" := "phi" + "w0c_16_23_4" * SIN(4 * 0.4 * "x") + "w0d_16_23_4" * COS(4 * 0.4 * "x");
    "phi" := "phi" + "w0c_16_23_5" * SIN(5 * 0.4 * "x") + "w0d_16_23_5" * COS(5 * 0.4 * "x");
    "phi" := "phi" + "w0c_16_23_6" * SIN(6 * 0.4 * "x") + "w0d_16_23_6" * COS(6 * 0.4 * "x");
    "acc" := "acc" + "phi";
    "x" := "feat_24";
    "phi" := "w0b_16_24" * "x" / (1.0 + EXP(-"x"));
    "phi" := "phi" + "w0c_16_24_1" * SIN(1 * 0.4 * "x") + "w0d_16_24_1" * COS(1 * 0.4 * "x");
    "phi" := "phi" + "w0c_16_24_2" * SIN(2 * 0.4 * "x") + "w0d_16_24_2" * COS(2 * 0.4 * "x");
    "phi" := "phi" + "w0c_16_24_3" * SIN(3 * 0.4 * "x") + "w0d_16_24_3" * COS(3 * 0.4 * "x");
    "phi" := "phi" + "w0c_16_24_4" * SIN(4 * 0.4 * "x") + "w0d_16_24_4" * COS(4 * 0.4 * "x");
    "phi" := "phi" + "w0c_16_24_5" * SIN(5 * 0.4 * "x") + "w0d_16_24_5" * COS(5 * 0.4 * "x");
    "phi" := "phi" + "w0c_16_24_6" * SIN(6 * 0.4 * "x") + "w0d_16_24_6" * COS(6 * 0.4 * "x");
    "acc" := "acc" + "phi";
    "x" := "feat_25";
    "phi" := "w0b_16_25" * "x" / (1.0 + EXP(-"x"));
    "phi" := "phi" + "w0c_16_25_1" * SIN(1 * 0.4 * "x") + "w0d_16_25_1" * COS(1 * 0.4 * "x");
    "phi" := "phi" + "w0c_16_25_2" * SIN(2 * 0.4 * "x") + "w0d_16_25_2" * COS(2 * 0.4 * "x");
    "phi" := "phi" + "w0c_16_25_3" * SIN(3 * 0.4 * "x") + "w0d_16_25_3" * COS(3 * 0.4 * "x");
    "phi" := "phi" + "w0c_16_25_4" * SIN(4 * 0.4 * "x") + "w0d_16_25_4" * COS(4 * 0.4 * "x");
    "phi" := "phi" + "w0c_16_25_5" * SIN(5 * 0.4 * "x") + "w0d_16_25_5" * COS(5 * 0.4 * "x");
    "phi" := "phi" + "w0c_16_25_6" * SIN(6 * 0.4 * "x") + "w0d_16_25_6" * COS(6 * 0.4 * "x");
    "acc" := "acc" + "phi";
    "x" := "feat_26";
    "phi" := "w0b_16_26" * "x" / (1.0 + EXP(-"x"));
    "phi" := "phi" + "w0c_16_26_1" * SIN(1 * 0.4 * "x") + "w0d_16_26_1" * COS(1 * 0.4 * "x");
    "phi" := "phi" + "w0c_16_26_2" * SIN(2 * 0.4 * "x") + "w0d_16_26_2" * COS(2 * 0.4 * "x");
    "phi" := "phi" + "w0c_16_26_3" * SIN(3 * 0.4 * "x") + "w0d_16_26_3" * COS(3 * 0.4 * "x");
    "phi" := "phi" + "w0c_16_26_4" * SIN(4 * 0.4 * "x") + "w0d_16_26_4" * COS(4 * 0.4 * "x");
    "phi" := "phi" + "w0c_16_26_5" * SIN(5 * 0.4 * "x") + "w0d_16_26_5" * COS(5 * 0.4 * "x");
    "phi" := "phi" + "w0c_16_26_6" * SIN(6 * 0.4 * "x") + "w0d_16_26_6" * COS(6 * 0.4 * "x");
    "acc" := "acc" + "phi";
    "x" := "feat_27";
    "phi" := "w0b_16_27" * "x" / (1.0 + EXP(-"x"));
    "phi" := "phi" + "w0c_16_27_1" * SIN(1 * 0.4 * "x") + "w0d_16_27_1" * COS(1 * 0.4 * "x");
    "phi" := "phi" + "w0c_16_27_2" * SIN(2 * 0.4 * "x") + "w0d_16_27_2" * COS(2 * 0.4 * "x");
    "phi" := "phi" + "w0c_16_27_3" * SIN(3 * 0.4 * "x") + "w0d_16_27_3" * COS(3 * 0.4 * "x");
    "phi" := "phi" + "w0c_16_27_4" * SIN(4 * 0.4 * "x") + "w0d_16_27_4" * COS(4 * 0.4 * "x");
    "phi" := "phi" + "w0c_16_27_5" * SIN(5 * 0.4 * "x") + "w0d_16_27_5" * COS(5 * 0.4 * "x");
    "phi" := "phi" + "w0c_16_27_6" * SIN(6 * 0.4 * "x") + "w0d_16_27_6" * COS(6 * 0.4 * "x");
    "acc" := "acc" + "phi";
    "x" := "feat_28";
    "phi" := "w0b_16_28" * "x" / (1.0 + EXP(-"x"));
    "phi" := "phi" + "w0c_16_28_1" * SIN(1 * 0.4 * "x") + "w0d_16_28_1" * COS(1 * 0.4 * "x");
    "phi" := "phi" + "w0c_16_28_2" * SIN(2 * 0.4 * "x") + "w0d_16_28_2" * COS(2 * 0.4 * "x");
    "phi" := "phi" + "w0c_16_28_3" * SIN(3 * 0.4 * "x") + "w0d_16_28_3" * COS(3 * 0.4 * "x");
    "phi" := "phi" + "w0c_16_28_4" * SIN(4 * 0.4 * "x") + "w0d_16_28_4" * COS(4 * 0.4 * "x");
    "phi" := "phi" + "w0c_16_28_5" * SIN(5 * 0.4 * "x") + "w0d_16_28_5" * COS(5 * 0.4 * "x");
    "phi" := "phi" + "w0c_16_28_6" * SIN(6 * 0.4 * "x") + "w0d_16_28_6" * COS(6 * 0.4 * "x");
    "acc" := "acc" + "phi";
    "h1_16" := "acc" + "b0_16";
    // === L1 (16->4): LUT N=16, domain [-3.15,3.15] ===
    // input 1: binary search on L1 grid
    "lo" := 0; "hi" := 15;
    "x" := "h1_1";
    IF "x" < -3.15 THEN "x" := -3.15; END_IF;
    IF "x" > 3.15 THEN "x" := 3.15; END_IF;
    WHILE "hi" - "lo" > 1 DO
        "mid" := "lo" + ("hi" - "lo") / 2;
        IF "x" > "g1_1"["mid"] THEN "lo" := "mid"; ELSE "hi" := "mid"; END_IF;
    END_WHILE;
    "t" := ("x" - "g1_1"["lo"]) / ("g1_1"["hi"] - "g1_1"["lo"] + 1.0E-10);
    "class_1" := "class_1" + ("t1_1_1"["lo"] * (1.0 - "t") + "t1_1_1"["hi"] * "t");
    "class_2" := "class_2" + ("t1_2_1"["lo"] * (1.0 - "t") + "t1_2_1"["hi"] * "t");
    "class_3" := "class_3" + ("t1_3_1"["lo"] * (1.0 - "t") + "t1_3_1"["hi"] * "t");
    "class_4" := "class_4" + ("t1_4_1"["lo"] * (1.0 - "t") + "t1_4_1"["hi"] * "t");
    // input 2: binary search on L1 grid
    "lo" := 0; "hi" := 15;
    "x" := "h1_2";
    IF "x" < -3.15 THEN "x" := -3.15; END_IF;
    IF "x" > 3.15 THEN "x" := 3.15; END_IF;
    WHILE "hi" - "lo" > 1 DO
        "mid" := "lo" + ("hi" - "lo") / 2;
        IF "x" > "g1_2"["mid"] THEN "lo" := "mid"; ELSE "hi" := "mid"; END_IF;
    END_WHILE;
    "t" := ("x" - "g1_2"["lo"]) / ("g1_2"["hi"] - "g1_2"["lo"] + 1.0E-10);
    "class_1" := "class_1" + ("t1_1_2"["lo"] * (1.0 - "t") + "t1_1_2"["hi"] * "t");
    "class_2" := "class_2" + ("t1_2_2"["lo"] * (1.0 - "t") + "t1_2_2"["hi"] * "t");
    "class_3" := "class_3" + ("t1_3_2"["lo"] * (1.0 - "t") + "t1_3_2"["hi"] * "t");
    "class_4" := "class_4" + ("t1_4_2"["lo"] * (1.0 - "t") + "t1_4_2"["hi"] * "t");
    // input 3: binary search on L1 grid
    "lo" := 0; "hi" := 15;
    "x" := "h1_3";
    IF "x" < -3.15 THEN "x" := -3.15; END_IF;
    IF "x" > 3.15 THEN "x" := 3.15; END_IF;
    WHILE "hi" - "lo" > 1 DO
        "mid" := "lo" + ("hi" - "lo") / 2;
        IF "x" > "g1_3"["mid"] THEN "lo" := "mid"; ELSE "hi" := "mid"; END_IF;
    END_WHILE;
    "t" := ("x" - "g1_3"["lo"]) / ("g1_3"["hi"] - "g1_3"["lo"] + 1.0E-10);
    "class_1" := "class_1" + ("t1_1_3"["lo"] * (1.0 - "t") + "t1_1_3"["hi"] * "t");
    "class_2" := "class_2" + ("t1_2_3"["lo"] * (1.0 - "t") + "t1_2_3"["hi"] * "t");
    "class_3" := "class_3" + ("t1_3_3"["lo"] * (1.0 - "t") + "t1_3_3"["hi"] * "t");
    "class_4" := "class_4" + ("t1_4_3"["lo"] * (1.0 - "t") + "t1_4_3"["hi"] * "t");
    // input 4: binary search on L1 grid
    "lo" := 0; "hi" := 15;
    "x" := "h1_4";
    IF "x" < -3.15 THEN "x" := -3.15; END_IF;
    IF "x" > 3.15 THEN "x" := 3.15; END_IF;
    WHILE "hi" - "lo" > 1 DO
        "mid" := "lo" + ("hi" - "lo") / 2;
        IF "x" > "g1_4"["mid"] THEN "lo" := "mid"; ELSE "hi" := "mid"; END_IF;
    END_WHILE;
    "t" := ("x" - "g1_4"["lo"]) / ("g1_4"["hi"] - "g1_4"["lo"] + 1.0E-10);
    "class_1" := "class_1" + ("t1_1_4"["lo"] * (1.0 - "t") + "t1_1_4"["hi"] * "t");
    "class_2" := "class_2" + ("t1_2_4"["lo"] * (1.0 - "t") + "t1_2_4"["hi"] * "t");
    "class_3" := "class_3" + ("t1_3_4"["lo"] * (1.0 - "t") + "t1_3_4"["hi"] * "t");
    "class_4" := "class_4" + ("t1_4_4"["lo"] * (1.0 - "t") + "t1_4_4"["hi"] * "t");
    // input 5: binary search on L1 grid
    "lo" := 0; "hi" := 15;
    "x" := "h1_5";
    IF "x" < -3.15 THEN "x" := -3.15; END_IF;
    IF "x" > 3.15 THEN "x" := 3.15; END_IF;
    WHILE "hi" - "lo" > 1 DO
        "mid" := "lo" + ("hi" - "lo") / 2;
        IF "x" > "g1_5"["mid"] THEN "lo" := "mid"; ELSE "hi" := "mid"; END_IF;
    END_WHILE;
    "t" := ("x" - "g1_5"["lo"]) / ("g1_5"["hi"] - "g1_5"["lo"] + 1.0E-10);
    "class_1" := "class_1" + ("t1_1_5"["lo"] * (1.0 - "t") + "t1_1_5"["hi"] * "t");
    "class_2" := "class_2" + ("t1_2_5"["lo"] * (1.0 - "t") + "t1_2_5"["hi"] * "t");
    "class_3" := "class_3" + ("t1_3_5"["lo"] * (1.0 - "t") + "t1_3_5"["hi"] * "t");
    "class_4" := "class_4" + ("t1_4_5"["lo"] * (1.0 - "t") + "t1_4_5"["hi"] * "t");
    // input 6: binary search on L1 grid
    "lo" := 0; "hi" := 15;
    "x" := "h1_6";
    IF "x" < -3.15 THEN "x" := -3.15; END_IF;
    IF "x" > 3.15 THEN "x" := 3.15; END_IF;
    WHILE "hi" - "lo" > 1 DO
        "mid" := "lo" + ("hi" - "lo") / 2;
        IF "x" > "g1_6"["mid"] THEN "lo" := "mid"; ELSE "hi" := "mid"; END_IF;
    END_WHILE;
